C01789=1024.573,0.095,-96.896,167.247,47.803,158.792
C01790=1024.568,-0.154,-96.882,167.244,47.807,158.792
C01791=1024.561,-0.404,-96.867,167.241,47.810,158.792
C01792=1024.555,-0.653,-96.854,167.239,47.813,158.792
C01793=1024.549,-0.902,-96.839,167.236,47.817,158.792
C01794=1024.543,-1.152,-96.825,167.234,47.820,158.793
C01795=1024.538,-1.401,-96.810,167.231,47.823,158.793
C01796=1024.532,-1.652,-96.796,167.228,47.826,158.793
C01797=1024.526,-1.901,-96.782,167.226,47.830,158.794
C01798=1024.520,-2.150,-96.768,167.223,47.833,158.794
C01799=1024.514,-2.400,-96.753,167.221,47.836,158.794
C01800=1024.508,-2.649,-96.739,167.218,47.840,158.794
C01801=1024.502,-2.899,-96.726,167.214,47.843,158.794
C01802=1024.496,-3.148,-96.711,167.212,47.846,158.795
C01803=1024.490,-3.398,-96.697,167.209,47.850,158.795
C01804=1024.484,-3.648,-96.683,167.206,47.853,158.795
C01805=1024.478,-3.897,-96.668,167.204,47.856,158.795
C01806=1024.473,-4.147,-96.654,167.201,47.860,158.796
C01807=1024.466,-4.429,-96.639,167.198,47.863,158.796
C01808=1024.458,-4.711,-96.623,167.196,47.867,158.796
C01809=1024.452,-4.993,-96.608,167.193,47.871,158.797
C01810=1024.444,-5.274,-96.592,167.189,47.875,158.797
C01811=1024.439,-5.524,-96.578,167.187,47.878,158.797
C01812=1024.433,-5.774,-96.564,167.184,47.882,158.797
C01813=1024.426,-6.024,-96.550,167.181,47.885,158.798
C01814=1024.421,-6.272,-96.536,167.179,47.889,158.798
C01815=1024.414,-6.522,-96.522,167.176,47.892,158.798
C01816=1024.408,-6.772,-96.508,167.173,47.896,158.798
C01817=1024.402,-7.021,-96.495,167.169,47.899,158.799
C01818=1024.397,-7.271,-96.481,167.168,47.903,158.799
C01819=1024.389,-7.520,-96.467,167.164,47.906,158.799
C01820=1024.384,-7.770,-96.453,167.162,47.910,158.800
C01821=1024.378,-8.019,-96.439,167.159,47.912,158.800
C01822=1024.372,-8.269,-96.425,167.157,47.916,158.800
C01823=1024.366,-8.519,-96.412,167.153,47.919,158.800
C01824=1024.360,-8.768,-96.398,167.151,47.923,158.801
C01825=1024.353,-9.018,-96.384,167.148,47.926,158.801
C01826=1024.348,-9.268,-96.371,167.146,47.930,158.801
C01827=1024.341,-9.516,-96.357,167.142,47.933,158.801
C01828=1024.336,-9.766,-96.343,167.141,47.937,158.802
C01829=1024.329,-10.016,-96.329,167.137,47.940,158.802
C01830=1024.323,-10.265,-96.315,167.134,47.943,158.802
C01831=1024.317,-10.515,-96.302,167.132,47.947,158.802
C01832=1024.312,-10.764,-96.288,167.129,47.950,158.802
C01833=1024.305,-11.014,-96.274,167.126,47.954,158.803
C01834=1024.299,-11.264,-96.261,167.123,47.957,158.803
C01835=1024.293,-11.513,-96.247,167.121,47.960,158.803
C01836=1024.288,-11.763,-96.233,167.118,47.964,158.804
C01837=1024.281,-12.013,-96.220,167.115,47.967,158.804
C01838=1024.275,-12.262,-96.206,167.113,47.970,158.804
C01839=1024.269,-12.511,-96.193,167.110,47.974,158.804
C01840=1024.264,-12.761,-96.179,167.107,47.977,158.805
C01841=1024.258,-13.010,-96.166,167.105,47.980,158.805
C01842=1024.252,-13.261,-96.151,167.102,47.984,158.805
C01843=1024.245,-13.510,-96.138,167.099,47.987,158.805
C01844=1024.240,-13.759,-96.124,167.096,47.991,158.805
C01845=1024.234,-14.009,-96.111,167.094,47.994,158.806
C01846=1024.228,-14.258,-96.097,167.091,47.997,158.806
C01847=1024.221,-14.508,-96.083,167.088,48.000,158.806
C01848=1024.216,-14.758,-96.070,167.086,48.004,158.806
C01849=1024.210,-15.007,-96.056,167.083,48.007,158.807
C01850=1024.204,-15.257,-96.042,167.080,48.011,158.807
C01851=1024.198,-15.506,-96.029,167.078,48.014,158.807
C01852=1024.192,-15.755,-96.015,167.074,48.017,158.807
C01853=1024.186,-16.005,-96.002,167.072,48.021,158.808
C01854=1024.180,-16.255,-95.989,167.068,48.024,158.808
C01855=1024.174,-16.505,-95.976,167.067,48.028,158.808
C01856=1024.167,-16.754,-95.963,167.063,48.031,158.808
C01857=1024.162,-17.003,-95.949,167.060,48.035,158.809
C01858=1024.156,-17.253,-95.935,167.057,48.038,158.809
C01859=1024.149,-17.503,-95.923,167.054,48.042,158.809
C01860=1024.143,-17.753,-95.909,167.052,48.045,158.809
C01861=1024.137,-18.002,-95.895,167.049,48.049,158.810
C01862=1024.131,-18.251,-95.882,167.046,48.052,158.810
C01863=1024.125,-18.501,-95.870,167.043,48.056,158.810
C01864=1024.119,-18.751,-95.856,167.041,48.059,158.810
C01865=1024.113,-19.000,-95.843,167.038,48.062,158.811
C01866=1024.107,-19.249,-95.829,167.035,48.066,158.811
C01867=1024.101,-19.500,-95.816,167.032,48.070,158.811
C01868=1024.095,-19.749,-95.803,167.030,48.072,158.811
C01869=1024.088,-19.998,-95.790,167.027,48.076,158.812
C01870=1024.083,-20.248,-95.777,167.024,48.079,158.812
C01871=1024.076,-20.529,-95.762,167.021,48.083,158.812
C01872=1024.069,-20.809,-95.747,167.019,48.087,158.812
C01873=1024.062,-21.089,-95.732,167.015,48.091,158.813
C01874=1024.056,-21.369,-95.717,167.012,48.095,158.813
C01875=1024.050,-21.619,-95.704,167.009,48.098,158.813
C01876=1024.044,-21.868,-95.691,167.007,48.102,158.813
C01877=1024.037,-22.118,-95.678,167.004,48.105,158.814
C01878=1024.032,-22.368,-95.665,167.001,48.109,158.814
C01879=1024.026,-22.617,-95.651,166.998,48.112,158.814
C01880=1024.020,-22.866,-95.638,166.994,48.115,158.814
C01881=1024.014,-23.116,-95.626,166.993,48.119,158.815
C01882=1024.008,-23.366,-95.612,166.989,48.122,158.815
C01883=1024.002,-23.616,-95.600,166.987,48.126,158.815
C01884=1023.996,-23.865,-95.586,166.983,48.129,158.815
C01885=1023.990,-24.115,-95.573,166.981,48.132,158.815
C01886=1023.984,-24.364,-95.560,166.978,48.136,158.816
C01887=1023.978,-24.613,-95.547,166.975,48.139,158.816
C01888=1023.972,-24.863,-95.534,166.972,48.143,158.816
C01889=1023.967,-25.113,-95.520,166.970,48.146,158.816
C01890=1023.961,-25.363,-95.508,166.967,48.149,158.817
C01891=1023.954,-25.612,-95.494,166.964,48.153,158.817
C01892=1023.949,-25.862,-95.482,166.961,48.156,158.817
C01893=1023.942,-26.111,-95.469,166.959,48.159,158.817
C01894=1023.937,-26.361,-95.456,166.956,48.163,158.818
C01895=1023.931,-26.611,-95.442,166.953,48.166,158.818
C01896=1023.925,-26.861,-95.430,166.950,48.170,158.818
C01897=1023.919,-27.110,-95.416,166.948,48.173,158.818
C01898=1023.913,-27.360,-95.404,166.945,48.176,158.818
C01899=1023.907,-27.609,-95.391,166.942,48.180,158.819
C01900=1023.901,-27.859,-95.378,166.939,48.183,158.819
C01901=1023.895,-28.107,-95.365,166.936,48.187,158.819
C01902=1023.889,-28.357,-95.353,166.933,48.190,158.819
C01903=1023.883,-28.607,-95.340,166.931,48.194,158.820
C01904=1023.877,-28.856,-95.327,166.928,48.197,158.820
C01905=1023.871,-29.106,-95.314,166.925,48.201,158.820
C01906=1023.865,-29.356,-95.302,166.922,48.204,158.820
C01907=1023.859,-29.605,-95.288,166.919,48.208,158.821
C01908=1023.852,-29.855,-95.276,166.916,48.211,158.821
C01909=1023.847,-30.105,-95.264,166.914,48.215,158.821
C01910=1023.841,-30.355,-95.251,166.911,48.218,158.821
C01911=1023.834,-30.604,-95.238,166.908,48.222,158.822
C01912=1023.829,-30.854,-95.225,166.905,48.225,158.822
C01913=1023.823,-31.104,-95.213,166.902,48.229,158.822
C01914=1023.817,-31.352,-95.200,166.899,48.232,158.822
C01915=1023.811,-31.602,-95.187,166.897,48.236,158.822
C01916=1023.805,-31.852,-95.175,166.894,48.239,158.823
C01917=1023.799,-32.102,-95.162,166.891,48.243,158.823
C01918=1023.792,-32.351,-95.150,166.888,48.246,158.823
C01919=1023.786,-32.601,-95.137,166.885,48.250,158.823
C01920=1023.781,-32.851,-95.125,166.882,48.253,158.824
C01921=1023.775,-33.100,-95.112,166.880,48.257,158.824
C01922=1023.769,-33.350,-95.100,166.877,48.260,158.824
C01923=1023.763,-33.599,-95.087,166.874,48.263,158.824
C01924=1023.757,-33.849,-95.074,166.871,48.267,158.824
C01925=1023.751,-34.099,-95.061,166.868,48.270,158.825
C01926=1023.745,-34.349,-95.049,166.865,48.274,158.825
C01927=1023.739,-34.598,-95.037,166.863,48.277,158.825
C01928=1023.733,-34.847,-95.024,166.860,48.281,158.825
C01929=1023.727,-35.097,-95.012,166.857,48.284,158.826
C01930=1023.721,-35.347,-94.999,166.853,48.288,158.826
C01931=1023.715,-35.597,-94.986,166.851,48.291,158.826
C01932=1023.710,-35.846,-94.974,166.847,48.295,158.826
C01933=1023.704,-36.096,-94.962,166.846,48.298,158.827
C01934=1023.698,-36.346,-94.949,166.842,48.302,158.827
C01935=1023.691,-36.625,-94.935,166.840,48.305,158.827
C01936=1023.685,-36.904,-94.921,166.836,48.310,158.827
C01937=1023.678,-37.184,-94.907,166.833,48.313,158.827
C01938=1023.671,-37.463,-94.893,166.830,48.317,158.828
C01939=1023.666,-37.712,-94.881,166.827,48.320,158.828
C01940=1023.660,-37.962,-94.869,166.824,48.324,158.828
C01941=1023.654,-38.212,-94.856,166.821,48.327,158.828
C01942=1023.648,-38.462,-94.844,166.818,48.331,158.828
C01943=1023.643,-38.711,-94.831,166.816,48.334,158.829
C01944=1023.636,-38.961,-94.819,166.812,48.337,158.829
C01945=1023.630,-39.210,-94.807,166.810,48.341,158.829
C01946=1023.624,-39.460,-94.794,166.806,48.344,158.829
C01947=1023.618,-39.709,-94.783,166.804,48.348,158.830
C01948=1023.612,-39.959,-94.770,166.800,48.351,158.830
C01949=1023.607,-40.209,-94.758,166.798,48.355,158.830
C01950=1023.600,-40.459,-94.746,166.794,48.358,158.830
C01951=1023.595,-40.708,-94.733,166.793,48.362,158.831
C01952=1023.589,-40.958,-94.721,166.789,48.365,158.831
C01953=1023.582,-41.207,-94.709,166.787,48.369,158.831
C01954=1023.577,-41.457,-94.697,166.783,48.372,158.831
C01955=1023.570,-41.707,-94.685,166.781,48.376,158.831
C01956=1023.565,-41.956,-94.673,166.777,48.379,158.832
C01957=1023.559,-42.206,-94.661,166.775,48.383,158.832
C01958=1023.553,-42.455,-94.649,166.771,48.387,158.832
C01959=1023.547,-42.705,-94.636,166.769,48.390,158.832
C01960=1023.541,-42.955,-94.625,166.765,48.394,158.832
C01961=1023.535,-43.204,-94.613,166.764,48.397,158.833
C01962=1023.529,-43.454,-94.600,166.761,48.401,158.833
C01963=1023.523,-43.703,-94.589,166.758,48.404,158.833
C01964=1023.517,-43.953,-94.576,166.755,48.408,158.833
C01965=1023.511,-44.203,-94.565,166.752,48.412,158.834
C01966=1023.505,-44.452,-94.553,166.749,48.415,158.834
C01967=1023.500,-44.702,-94.540,166.746,48.419,158.834
C01968=1023.493,-44.952,-94.528,166.743,48.422,158.834
C01969=1023.488,-45.202,-94.517,166.739,48.425,158.834
C01970=1023.481,-45.451,-94.505,166.737,48.429,158.835
C01971=1023.476,-45.700,-94.493,166.734,48.432,158.835
C01972=1023.470,-45.950,-94.480,166.732,48.436,158.835
C01973=1023.464,-46.201,-94.469,166.728,48.439,158.835
C01974=1023.458,-46.450,-94.457,166.726,48.443,158.836
C01975=1023.452,-46.699,-94.445,166.722,48.446,158.836
C01976=1023.447,-46.949,-94.433,166.719,48.449,158.836
C01977=1023.440,-47.199,-94.421,166.716,48.453,158.836
C01978=1023.435,-47.448,-94.409,166.713,48.457,158.836
C01979=1023.429,-47.698,-94.396,166.710,48.461,158.837
C01980=1023.423,-47.947,-94.386,166.708,48.463,158.837
C01981=1023.417,-48.197,-94.373,166.705,48.467,158.837
C01982=1023.411,-48.447,-94.362,166.702,48.471,158.837
C01983=1023.406,-48.696,-94.350,166.699,48.474,158.837
C01984=1023.399,-48.946,-94.338,166.696,48.478,158.838
C01985=1023.394,-49.196,-94.326,166.693,48.481,158.838
C01986=1023.388,-49.446,-94.314,166.690,48.484,158.838
C01987=1023.382,-49.695,-94.302,166.687,48.488,158.838
C01988=1023.376,-49.945,-94.290,166.684,48.491,158.838
C01989=1023.370,-50.194,-94.279,166.682,48.494,158.839
C01990=1023.365,-50.444,-94.267,166.679,48.498,158.839
C01991=1023.359,-50.693,-94.255,166.676,48.501,158.839
C01992=1023.353,-50.944,-94.243,166.673,48.505,158.839
C01993=1023.347,-51.193,-94.232,166.670,48.509,158.839
C01994=1023.341,-51.443,-94.220,166.667,48.512,158.840
C01995=1023.335,-51.692,-94.209,166.664,48.516,158.840
C01996=1023.329,-51.942,-94.197,166.661,48.520,158.840
C01997=1023.323,-52.192,-94.186,166.658,48.524,158.840
C01998=1023.317,-52.441,-94.174,166.655,48.527,158.840
C01999=1023.310,-52.722,-94.162,166.652,48.532,158.841
C02000=1023.303,-53.001,-94.149,166.649,48.536,158.841
C02001=1023.297,-53.280,-94.136,166.645,48.540,158.841
C02002=1023.290,-53.561,-94.124,166.642,48.544,158.842
C02003=1023.284,-53.810,-94.112,166.639,48.547,158.842
C02004=1023.278,-54.060,-94.101,166.636,48.551,158.842
C02005=1023.272,-54.310,-94.089,166.633,48.554,158.842
C02006=1023.266,-54.559,-94.077,166.630,48.558,158.842
C02007=1023.261,-54.809,-94.066,166.627,48.562,158.843
C02008=1023.254,-55.059,-94.055,166.624,48.565,158.843
C02009=1023.248,-55.308,-94.044,166.621,48.569,158.843
C02010=1023.242,-55.558,-94.032,166.618,48.572,158.843
C02011=1023.236,-55.807,-94.021,166.615,48.576,158.844
C02012=1023.230,-56.058,-94.010,166.613,48.580,158.844
C02013=1023.224,-56.307,-93.998,166.609,48.583,158.844
C02014=1023.219,-56.556,-93.987,166.607,48.587,158.844
C02015=1023.212,-56.806,-93.976,166.603,48.591,158.844
C02016=1023.207,-57.056,-93.965,166.601,48.595,158.845
C02017=1023.200,-57.305,-93.953,166.597,48.598,158.845
C02018=1023.195,-57.555,-93.942,166.595,48.602,158.845
C02019=1023.189,-57.805,-93.931,166.591,48.605,158.845
C02020=1023.183,-58.055,-93.919,166.589,48.609,158.846
C02021=1023.177,-58.304,-93.908,166.585,48.612,158.846
C02022=1023.171,-58.553,-93.897,166.583,48.616,158.846
C02023=1023.165,-58.803,-93.886,166.580,48.620,158.846
C02024=1023.159,-59.053,-93.875,166.577,48.623,158.846
C02025=1023.153,-59.303,-93.863,166.574,48.627,158.847
C02026=1023.148,-59.553,-93.852,166.571,48.630,158.847
C02027=1023.142,-59.802,-93.841,166.568,48.634,158.847
C02028=1023.136,-60.051,-93.830,166.565,48.638,158.847
C02029=1023.130,-60.301,-93.818,166.562,48.642,158.847
C02030=1023.124,-60.551,-93.808,166.559,48.645,158.848
C02031=1023.118,-60.800,-93.797,166.556,48.649,158.848
C02032=1023.112,-61.051,-93.785,166.553,48.652,158.848
C02033=1023.107,-61.300,-93.774,166.550,48.656,158.848
C02034=1023.101,-61.550,-93.763,166.547,48.659,158.848
C02035=1023.095,-61.800,-93.752,166.544,48.663,158.849
C02036=1023.089,-62.050,-93.741,166.541,48.666,158.849
///RCONF 1,0,0,1,0,0,0,0,0,0,0,0,0,0,0,0,0,0,0,0,0,0,0,0
C02037=1023.083,-62.298,-93.729,166.538,48.670,158.849
C02038=1023.077,-62.548,-93.719,166.535,48.674,158.849
C02039=1023.072,-62.798,-93.707,166.532,48.677,158.849
C02040=1023.066,-63.048,-93.696,166.529,48.681,158.850
C02041=1023.060,-63.297,-93.685,166.526,48.684,158.850
C02042=1023.054,-63.547,-93.674,166.523,48.688,158.850
C02043=1023.048,-63.797,-93.663,166.520,48.691,158.850
C02044=1023.042,-64.047,-93.652,166.517,48.695,158.850
C02045=1023.036,-64.296,-93.641,166.514,48.698,158.851
C02046=1023.031,-64.546,-93.630,166.511,48.702,158.851
C02047=1023.025,-64.796,-93.618,166.508,48.705,158.851
C02048=1023.019,-65.046,-93.607,166.505,48.709,158.851
C02049=1023.014,-65.295,-93.597,166.502,48.713,158.851
C02050=1023.008,-65.545,-93.586,166.499,48.716,158.851
C02051=1023.002,-65.794,-93.575,166.496,48.720,158.852
C02052=1022.996,-66.044,-93.564,166.493,48.723,158.852
C02053=1022.990,-66.294,-93.553,166.490,48.727,158.852
C02054=1022.985,-66.544,-93.543,166.487,48.730,158.852
C02055=1022.980,-66.794,-93.531,166.484,48.734,158.852
C02056=1022.974,-67.043,-93.520,166.481,48.738,158.853
C02057=1022.968,-67.293,-93.509,166.478,48.741,158.853
C02058=1022.962,-67.542,-93.498,166.475,48.745,158.853
C02059=1022.956,-67.792,-93.487,166.472,48.748,158.853
C02060=1022.950,-68.042,-93.476,166.470,48.751,158.853
C02061=1022.945,-68.291,-93.465,166.467,48.755,158.854
C02062=1022.939,-68.541,-93.455,166.464,48.758,158.854
C02063=1022.933,-68.822,-93.443,166.460,48.762,158.854
C02064=1022.926,-69.104,-93.430,166.457,48.766,158.854
C02065=1022.920,-69.384,-93.418,166.453,48.771,158.854
C02066=1022.914,-69.665,-93.406,166.450,48.774,158.855
C02067=1022.908,-69.914,-93.395,166.447,48.778,158.855
C02068=1022.902,-70.164,-93.384,166.444,48.781,158.855
C02069=1022.896,-70.413,-93.374,166.441,48.785,158.855
C02070=1022.891,-70.663,-93.362,166.438,48.788,158.855
C02071=1022.886,-70.913,-93.352,166.435,48.791,158.855
C02072=1022.880,-71.163,-93.341,166.432,48.795,158.856
C02073=1022.874,-71.413,-93.330,166.429,48.799,158.856
C02074=1022.868,-71.662,-93.319,166.426,48.802,158.856
C02075=1022.863,-71.913,-93.309,166.423,48.806,158.856
C02076=1022.857,-72.162,-93.298,166.420,48.809,158.856
C02077=1022.851,-72.412,-93.287,166.417,48.812,158.856
C02078=1022.845,-72.661,-93.276,166.414,48.816,158.857
C02079=1022.840,-72.911,-93.266,166.411,48.820,158.857
C02080=1022.834,-73.161,-93.255,166.408,48.823,158.857
C02081=1022.829,-73.410,-93.244,166.405,48.827,158.857
C02082=1022.824,-73.660,-93.233,166.402,48.830,158.857
C02083=1022.818,-73.910,-93.223,166.398,48.833,158.857
C02084=1022.812,-74.160,-93.212,166.396,48.837,158.858
C02085=1022.807,-74.410,-93.202,166.394,48.840,158.858
C02086=1022.801,-74.659,-93.191,166.389,48.844,158.858
C02087=1022.795,-74.908,-93.180,166.387,48.848,158.858
C02088=1022.789,-75.158,-93.170,166.383,48.851,158.858
C02089=1022.784,-75.408,-93.159,166.381,48.855,158.859
C02090=1022.778,-75.658,-93.149,166.377,48.858,158.859
C02091=1022.772,-75.907,-93.139,166.375,48.862,158.859
C02092=1022.766,-76.157,-93.129,166.371,48.865,158.859
C02093=1022.760,-76.407,-93.118,166.369,48.869,158.859
C02094=1022.755,-76.657,-93.108,166.366,48.873,158.860
C02095=1022.749,-76.906,-93.097,166.363,48.877,158.860
C02096=1022.743,-77.156,-93.087,166.360,48.880,158.860
C02097=1022.737,-77.406,-93.076,166.357,48.884,158.860
C02098=1022.732,-77.656,-93.066,166.354,48.887,158.860
C02099=1022.726,-77.905,-93.055,166.351,48.891,158.861
C02100=1022.721,-78.155,-93.045,166.348,48.894,158.861
C02101=1022.715,-78.405,-93.036,166.345,48.898,158.861
C02102=1022.709,-78.654,-93.025,166.342,48.902,158.861
C02103=1022.704,-78.904,-93.015,166.339,48.906,158.861
C02104=1022.698,-79.154,-93.004,166.336,48.909,158.861
C02105=1022.692,-79.403,-92.994,166.333,48.913,158.862
C02106=1022.686,-79.653,-92.984,166.330,48.916,158.862
C02107=1022.681,-79.903,-92.973,166.327,48.920,158.862
C02108=1022.676,-80.153,-92.963,166.324,48.923,158.862
C02109=1022.669,-80.402,-92.953,166.320,48.928,158.862
C02110=1022.664,-80.652,-92.943,166.317,48.931,158.863
C02111=1022.657,-80.902,-92.933,166.314,48.935,158.863
C02112=1022.652,-81.152,-92.923,166.311,48.939,158.863
C02113=1022.646,-81.401,-92.913,166.308,48.942,158.863
C02114=1022.641,-81.651,-92.903,166.305,48.946,158.863
C02115=1022.635,-81.901,-92.893,166.302,48.949,158.864
C02116=1022.629,-82.151,-92.883,166.299,48.953,158.864
C02117=1022.623,-82.401,-92.874,166.297,48.957,158.864
C02118=1022.617,-82.650,-92.863,166.292,48.961,158.864
C02119=1022.611,-82.900,-92.853,166.290,48.965,158.864
C02120=1022.606,-83.149,-92.844,166.286,48.968,158.864
C02121=1022.600,-83.399,-92.834,166.284,48.972,158.865
C02122=1022.595,-83.649,-92.824,166.281,48.976,158.865
C02123=1022.588,-83.898,-92.813,166.278,48.979,158.865
C02124=1022.583,-84.148,-92.803,166.275,48.983,158.865
C02125=1022.576,-84.398,-92.794,166.272,48.987,158.866
C02126=1022.572,-84.648,-92.784,166.269,48.991,158.866
C02127=1022.565,-84.931,-92.773,166.265,48.995,158.866
C02128=1022.558,-85.214,-92.762,166.261,48.999,158.866
C02129=1022.551,-85.497,-92.751,166.258,49.003,158.866
C02130=1022.546,-85.780,-92.739,166.255,49.007,158.867
C02131=1022.539,-86.030,-92.729,166.252,49.011,158.867
C02132=1022.534,-86.280,-92.719,166.249,49.015,158.867
C02133=1022.528,-86.529,-92.710,166.246,49.019,158.867
C02134=1022.523,-86.779,-92.700,166.243,49.022,158.867
C02135=1022.517,-87.029,-92.690,166.239,49.026,158.868
C02136=1022.511,-87.279,-92.680,166.236,49.030,158.868
C02137=1022.506,-87.528,-92.671,166.233,49.033,158.868
C02138=1022.500,-87.778,-92.661,166.230,49.037,158.868
C02139=1022.494,-88.028,-92.651,166.227,49.041,158.868
C02140=1022.488,-88.278,-92.641,166.224,49.045,158.869
C02141=1022.483,-88.527,-92.632,166.221,49.048,158.869
C02142=1022.477,-88.777,-92.622,166.218,49.052,158.869
C02143=1022.472,-89.027,-92.612,166.215,49.055,158.869
C02144=1022.466,-89.276,-92.603,166.212,49.059,158.869
C02145=1022.461,-89.526,-92.593,166.209,49.062,158.869
C02146=1022.454,-89.776,-92.583,166.205,49.067,158.870
C02147=1022.449,-90.026,-92.573,166.202,49.070,158.870
C02148=1022.443,-90.275,-92.564,166.199,49.074,158.870
C02149=1022.438,-90.525,-92.553,166.196,49.077,158.870
C02150=1022.432,-90.775,-92.544,166.193,49.081,158.870
C02151=1022.427,-91.024,-92.534,166.190,49.085,158.870
C02152=1022.421,-91.274,-92.525,166.188,49.089,158.871
C02153=1022.415,-91.524,-92.514,166.184,49.092,158.871
C02154=1022.410,-91.773,-92.505,166.182,49.096,158.871
C02155=1022.404,-92.024,-92.496,166.178,49.099,158.871
C02156=1022.399,-92.273,-92.487,166.176,49.103,158.871
C02157=1022.393,-92.523,-92.477,166.173,49.106,158.871
C02158=1022.387,-92.773,-92.467,166.170,49.110,158.872
C02159=1022.382,-93.022,-92.458,166.166,49.114,158.872
C02160=1022.376,-93.272,-92.447,166.163,49.118,158.872
C02161=1022.371,-93.521,-92.438,166.160,49.121,158.872
C02162=1022.365,-93.772,-92.428,166.157,49.125,158.872
C02163=1022.360,-94.022,-92.419,166.154,49.129,158.872
C02164=1022.354,-94.271,-92.410,166.151,49.133,158.873
C02165=1022.349,-94.521,-92.400,166.148,49.136,158.873
C02166=1022.343,-94.770,-92.391,166.145,49.140,158.873
C02167=1022.338,-95.020,-92.381,166.142,49.143,158.873
C02168=1022.332,-95.270,-92.372,166.139,49.146,158.873
C02169=1022.327,-95.520,-92.362,166.136,49.150,158.874
C02170=1022.321,-95.770,-92.352,166.133,49.154,158.874
C02171=1022.316,-96.019,-92.343,166.130,49.158,158.874
C02172=1022.310,-96.270,-92.334,166.127,49.161,158.874
C02173=1022.304,-96.519,-92.324,166.124,49.165,158.874
C02174=1022.299,-96.769,-92.314,166.121,49.168,158.874
C02175=1022.293,-97.018,-92.305,166.117,49.172,158.874
C02176=1022.288,-97.269,-92.296,166.114,49.176,158.875
C02177=1022.283,-97.518,-92.286,166.111,49.179,158.875
C02178=1022.277,-97.768,-92.276,166.108,49.183,158.875
C02179=1022.272,-98.018,-92.268,166.105,49.186,158.875
C02180=1022.266,-98.268,-92.258,166.102,49.190,158.875
C02181=1022.260,-98.517,-92.249,166.099,49.194,158.876
C02182=1022.254,-98.767,-92.240,166.096,49.198,158.876
C02183=1022.249,-99.016,-92.231,166.093,49.202,158.876
C02184=1022.244,-99.267,-92.222,166.089,49.205,158.876
C02185=1022.238,-99.516,-92.212,166.086,49.209,158.876
C02186=1022.232,-99.766,-92.203,166.084,49.213,158.877
C02187=1022.227,-100.016,-92.194,166.081,49.217,158.877
C02188=1022.221,-100.266,-92.185,166.078,49.221,158.877
C02189=1022.215,-100.515,-92.176,166.075,49.224,158.877
C02190=1022.209,-100.765,-92.167,166.072,49.228,158.877
C02191=1022.204,-101.050,-92.157,166.068,49.232,158.877
C02192=1022.197,-101.336,-92.147,166.064,49.237,158.878
C02193=1022.191,-101.620,-92.136,166.061,49.241,158.878
C02194=1022.184,-101.906,-92.126,166.058,49.245,158.878
C02195=1022.179,-102.155,-92.116,166.055,49.249,158.878
C02196=1022.174,-102.405,-92.108,166.052,49.252,158.878
C02197=1022.168,-102.655,-92.098,166.048,49.256,158.879
C02198=1022.163,-102.904,-92.090,166.045,49.260,158.879
C02199=1022.156,-103.154,-92.080,166.042,49.264,158.879
C02200=1022.151,-103.404,-92.071,166.039,49.268,158.879
C02201=1022.146,-103.654,-92.063,166.036,49.271,158.879
C02202=1022.140,-103.904,-92.053,166.033,49.275,158.879
C02203=1022.135,-104.153,-92.044,166.030,49.278,158.880
C02204=1022.129,-104.403,-92.035,166.027,49.282,158.880
C02205=1022.124,-104.653,-92.026,166.024,49.286,158.880
C02206=1022.118,-104.903,-92.018,166.020,49.290,158.880
C02207=1022.112,-105.152,-92.008,166.017,49.294,158.880
C02208=1022.107,-105.402,-92.000,166.014,49.297,158.880
C02209=1022.102,-105.652,-91.991,166.012,49.301,158.881
C02210=1022.096,-105.902,-91.982,166.008,49.305,158.881
C02211=1022.091,-106.152,-91.973,166.006,49.309,158.881
C02212=1022.086,-106.401,-91.964,166.003,49.312,158.881
C02213=1022.080,-106.651,-91.955,166.000,49.316,158.881
C02214=1022.074,-106.901,-91.946,165.996,49.320,158.881
C02215=1022.069,-107.151,-91.938,165.993,49.324,158.882
C02216=1022.063,-107.401,-91.929,165.990,49.328,158.882
C02217=1022.058,-107.650,-91.920,165.987,49.331,158.882
C02218=1022.052,-107.900,-91.911,165.984,49.335,158.882
C02219=1022.047,-108.150,-91.902,165.981,49.338,158.882
C02220=1022.041,-108.400,-91.894,165.978,49.342,158.883
C02221=1022.036,-108.650,-91.885,165.975,49.346,158.883
C02222=1022.030,-108.899,-91.876,165.971,49.350,158.883
C02223=1022.025,-109.149,-91.867,165.968,49.354,158.883
C02224=1022.019,-109.399,-91.859,165.965,49.357,158.883
C02225=1022.013,-109.648,-91.851,165.963,49.361,158.883
C02226=1022.008,-109.898,-91.842,165.960,49.365,158.884
C02227=1022.002,-110.149,-91.833,165.957,49.369,158.884
C02228=1021.997,-110.398,-91.824,165.953,49.373,158.884
C02229=1021.991,-110.647,-91.816,165.950,49.377,158.884
C02230=1021.986,-110.897,-91.807,165.947,49.380,158.884
C02231=1021.980,-111.147,-91.798,165.944,49.384,158.885
C02232=1021.975,-111.397,-91.790,165.941,49.388,158.885
C02233=1021.970,-111.647,-91.781,165.938,49.392,158.885
C02234=1021.964,-111.897,-91.773,165.935,49.396,158.885
C02235=1021.959,-112.146,-91.765,165.932,49.399,158.885
C02236=1021.953,-112.397,-91.756,165.928,49.403,158.885
C02237=1021.947,-112.646,-91.748,165.925,49.407,158.885
C02238=1021.942,-112.896,-91.739,165.923,49.411,158.886
C02239=1021.937,-113.146,-91.731,165.919,49.414,158.886
C02240=1021.931,-113.395,-91.722,165.917,49.418,158.886
C02241=1021.926,-113.646,-91.713,165.914,49.422,158.886
C02242=1021.920,-113.895,-91.705,165.911,49.425,158.886
C02243=1021.915,-114.145,-91.697,165.907,49.430,158.887
C02244=1021.910,-114.395,-91.688,165.904,49.433,158.887
C02245=1021.905,-114.645,-91.680,165.901,49.437,158.887
C02246=1021.899,-114.894,-91.672,165.898,49.441,158.887
C02247=1021.893,-115.144,-91.663,165.895,49.444,158.887
C02248=1021.887,-115.394,-91.654,165.892,49.448,158.888
C02249=1021.882,-115.644,-91.646,165.890,49.452,158.888
C02250=1021.877,-115.894,-91.637,165.885,49.456,158.888
C02251=1021.871,-116.143,-91.629,165.883,49.460,158.888
C02252=1021.866,-116.393,-91.621,165.879,49.463,158.888
C02253=1021.860,-116.642,-91.612,165.877,49.467,158.888
C02254=1021.855,-116.893,-91.605,165.874,49.471,158.889
C02255=1021.849,-117.178,-91.595,165.870,49.476,158.889
C02256=1021.843,-117.462,-91.586,165.866,49.480,158.889
C02257=1021.837,-117.747,-91.576,165.863,49.484,158.889
C02258=1021.830,-118.032,-91.567,165.860,49.488,158.889
C02259=1021.824,-118.282,-91.559,165.857,49.493,158.890
C02260=1021.819,-118.531,-91.550,165.854,49.497,158.890
C02261=1021.814,-118.782,-91.542,165.850,49.500,158.890
C02262=1021.809,-119.031,-91.534,165.847,49.504,158.890
C02263=1021.803,-119.281,-91.526,165.844,49.508,158.890
C02264=1021.798,-119.530,-91.518,165.841,49.512,158.890
C02265=1021.793,-119.781,-91.510,165.838,49.516,158.891
C02266=1021.787,-120.030,-91.502,165.835,49.519,158.891
C02267=1021.781,-120.280,-91.493,165.833,49.523,158.891
C02268=1021.776,-120.530,-91.485,165.829,49.527,158.891
C02269=1021.771,-120.780,-91.477,165.826,49.531,158.891
C02270=1021.765,-121.029,-91.469,165.823,49.535,158.891
C02271=1021.760,-121.279,-91.461,165.820,49.538,158.891
C02272=1021.755,-121.529,-91.453,165.817,49.542,158.892
C02273=1021.749,-121.779,-91.445,165.814,49.546,158.892
C02274=1021.744,-122.029,-91.437,165.811,49.549,158.892
C02275=1021.739,-122.279,-91.429,165.807,49.554,158.892
C02276=1021.733,-122.528,-91.421,165.804,49.558,158.892
C02277=1021.727,-122.778,-91.412,165.801,49.561,158.893
C02278=1021.722,-123.028,-91.405,165.799,49.565,158.893
C02279=1021.716,-123.278,-91.397,165.795,49.569,158.893
C02280=1021.711,-123.527,-91.388,165.793,49.573,158.893
C02281=1021.706,-123.778,-91.381,165.790,49.577,158.893
C02282=1021.700,-124.027,-91.373,165.787,49.580,158.893
C02283=1021.695,-124.278,-91.365,165.783,49.584,158.894
C02284=1021.690,-124.527,-91.356,165.780,49.588,158.894
C02285=1021.684,-124.777,-91.349,165.777,49.592,158.894
C02286=1021.679,-125.027,-91.341,165.774,49.596,158.894
C02287=1021.673,-125.276,-91.333,165.772,49.600,158.894
C02288=1021.668,-125.527,-91.325,165.768,49.603,158.895
C02289=1021.662,-125.776,-91.317,165.765,49.607,158.895
C02290=1021.658,-126.026,-91.310,165.762,49.612,158.895
C02291=1021.652,-126.276,-91.303,165.759,49.615,158.895
C02292=1021.647,-126.526,-91.294,165.756,49.619,158.895
C02293=1021.642,-126.776,-91.286,165.753,49.623,158.895
C02294=1021.636,-127.025,-91.278,165.750,49.626,158.896
C02295=1021.631,-127.276,-91.271,165.747,49.630,158.896
C02296=1021.625,-127.525,-91.263,165.743,49.635,158.896
C02297=1021.621,-127.775,-91.255,165.740,49.638,158.896
C02298=1021.615,-128.024,-91.248,165.738,49.642,158.896
C02299=1021.609,-128.274,-91.239,165.734,49.645,158.896
C02300=1021.605,-128.523,-91.230,165.732,49.648,158.897
C02301=1021.601,-128.773,-91.221,165.729,49.650,158.896
C02302=1021.598,-129.022,-91.211,165.726,49.653,158.896
C02303=1021.595,-129.272,-91.200,165.723,49.654,158.896
C02304=1021.592,-129.522,-91.189,165.721,49.655,158.896
C02305=1021.591,-129.772,-91.177,165.719,49.655,158.895
C02306=1021.589,-130.021,-91.165,165.716,49.655,158.895
C02307=1021.588,-130.271,-91.153,165.714,49.654,158.895
C02308=1021.587,-130.521,-91.138,165.711,49.653,158.894
C02309=1021.587,-130.771,-91.124,165.709,49.652,158.893
C02310=1021.588,-131.020,-91.110,165.707,49.649,158.893
C02311=1021.588,-131.270,-91.095,165.705,49.646,158.892
C02312=1021.590,-131.520,-91.078,165.703,49.644,158.891
C02313=1021.592,-131.770,-91.062,165.701,49.640,158.890
C02314=1021.594,-132.019,-91.046,165.700,49.635,158.889
C02315=1021.597,-132.269,-91.028,165.698,49.630,158.888
C02316=1021.600,-132.520,-91.009,165.696,49.625,158.887
C02317=1021.604,-132.769,-90.990,165.695,49.620,158.886
C02318=1021.608,-133.018,-90.971,165.693,49.614,158.884
C02319=1021.324,-133.044,-91.324,165.647,49.915,158.928
C02320=1021.321,-132.937,-91.332,165.648,49.918,158.929
C02321=1021.316,-132.580,-91.360,165.650,49.927,158.931
C02322=1021.313,-132.330,-91.378,165.651,49.932,158.932
C02323=1021.310,-132.080,-91.396,165.652,49.937,158.933
C02324=1021.308,-131.830,-91.413,165.655,49.941,158.934
C02325=1021.305,-131.580,-91.429,165.656,49.945,158.935
C02326=1021.304,-131.331,-91.445,165.659,49.948,158.936
C02327=1021.303,-131.081,-91.461,165.661,49.951,158.936
C02328=1021.302,-130.831,-91.475,165.663,49.953,158.937
C02329=1021.303,-130.581,-91.490,165.665,49.955,158.938
C02330=1021.304,-130.332,-91.503,165.667,49.956,158.938
C02331=1021.305,-130.082,-91.516,165.669,49.957,158.939
C02332=1021.305,-129.832,-91.528,165.672,49.957,158.939
C02333=1021.309,-129.420,-91.548,165.676,49.956,158.940
C02334=1021.313,-129.008,-91.565,165.680,49.954,158.940
C02335=1021.320,-128.596,-91.582,165.685,49.950,158.940
C02336=1021.327,-128.185,-91.596,165.690,49.946,158.940
C02337=1021.332,-127.935,-91.604,165.693,49.942,158.940
C02338=1021.338,-127.685,-91.612,165.696,49.938,158.940
C02339=1021.343,-127.435,-91.620,165.699,49.934,158.940
C02340=1021.348,-127.186,-91.627,165.701,49.930,158.939
C02341=1021.353,-126.936,-91.635,165.706,49.926,158.939
C02342=1021.359,-126.687,-91.643,165.708,49.922,158.939
C02343=1021.364,-126.436,-91.651,165.711,49.918,158.939
C02344=1021.370,-126.187,-91.658,165.714,49.914,158.939
C02345=1021.375,-125.936,-91.666,165.717,49.911,158.939
C02346=1021.381,-125.688,-91.674,165.721,49.906,158.939
C02347=1021.386,-125.437,-91.681,165.723,49.902,158.938
C02348=1021.391,-125.187,-91.689,165.726,49.898,158.938
C02349=1021.397,-124.938,-91.697,165.729,49.895,158.938
C02350=1021.402,-124.688,-91.704,165.732,49.891,158.938
C02351=1021.408,-124.438,-91.713,165.736,49.886,158.938
C02352=1021.413,-124.188,-91.721,165.739,49.883,158.938
C02353=1021.419,-123.938,-91.728,165.742,49.879,158.937
C02354=1021.424,-123.689,-91.737,165.744,49.875,158.937
C02355=1021.429,-123.438,-91.745,165.748,49.872,158.937
C02356=1021.434,-123.190,-91.752,165.750,49.868,158.937
C02357=1021.439,-122.939,-91.760,165.754,49.863,158.937
C02358=1021.444,-122.689,-91.768,165.757,49.860,158.936
C02359=1021.450,-122.440,-91.776,165.760,49.856,158.936
C02360=1021.455,-122.190,-91.784,165.763,49.852,158.936
C02361=1021.461,-121.940,-91.793,165.766,49.848,158.936
C02362=1021.467,-121.691,-91.801,165.769,49.844,158.936
C02363=1021.472,-121.440,-91.808,165.772,49.840,158.936
C02364=1021.477,-121.191,-91.817,165.775,49.837,158.935
C02365=1021.483,-120.941,-91.825,165.778,49.832,158.935
C02366=1021.488,-120.691,-91.832,165.781,49.828,158.935
C02367=1021.493,-120.441,-91.841,165.784,49.825,158.935
C02368=1021.499,-120.192,-91.849,165.787,49.821,158.935
C02369=1021.504,-119.941,-91.857,165.791,49.817,158.934
C02370=1021.509,-119.692,-91.865,165.794,49.813,158.934
C02371=1021.515,-119.442,-91.874,165.796,49.809,158.934
C02372=1021.521,-119.193,-91.881,165.799,49.805,158.934
C02373=1021.526,-118.942,-91.889,165.802,49.801,158.934
C02374=1021.531,-118.692,-91.898,165.806,49.797,158.934
C02375=1021.536,-118.443,-91.906,165.809,49.793,158.933
C02376=1021.542,-118.193,-91.914,165.812,49.789,158.933
C02377=1021.549,-117.874,-91.924,165.815,49.785,158.933
C02378=1021.556,-117.555,-91.935,165.820,49.779,158.933
C02379=1021.563,-117.238,-91.945,165.823,49.774,158.933
C02380=1021.570,-116.919,-91.956,165.827,49.770,158.932
C02381=1021.575,-116.669,-91.965,165.831,49.766,158.932
C02382=1021.580,-116.419,-91.972,165.834,49.762,158.932
C02383=1021.586,-116.170,-91.980,165.837,49.758,158.932
C02384=1021.591,-115.920,-91.989,165.839,49.754,158.932
C02385=1021.596,-115.670,-91.997,165.842,49.750,158.931
C02386=1021.602,-115.420,-92.006,165.845,49.747,158.931
C02387=1021.608,-115.171,-92.014,165.849,49.742,158.931
C02388=1021.614,-114.921,-92.023,165.852,49.738,158.931
C02389=1021.619,-114.671,-92.031,165.855,49.734,158.931
C02390=1021.624,-114.421,-92.040,165.858,49.731,158.931
C02391=1021.629,-114.171,-92.047,165.860,49.727,158.930
C02392=1021.634,-113.921,-92.056,165.865,49.723,158.930
C02393=1021.640,-113.671,-92.064,165.867,49.719,158.930
C02394=1021.645,-113.422,-92.073,165.870,49.715,158.930
C02395=1021.651,-113.172,-92.081,165.873,49.712,158.930
C02396=1021.657,-112.922,-92.089,165.876,49.708,158.929
C02397=1021.662,-112.672,-92.098,165.879,49.704,158.929
C02398=1021.667,-112.422,-92.106,165.883,49.700,158.929
C02399=1021.672,-112.173,-92.115,165.886,49.696,158.929
C02400=1021.678,-111.924,-92.124,165.888,49.692,158.929
C02401=1021.684,-111.673,-92.133,165.892,49.689,158.929
C02402=1021.689,-111.423,-92.141,165.894,49.685,158.928
C02403=1021.694,-111.174,-92.150,165.897,49.681,158.928
C02404=1021.700,-110.924,-92.158,165.901,49.677,158.928
C02405=1021.705,-110.674,-92.167,165.904,49.673,158.928
C02406=1021.712,-110.424,-92.175,165.907,49.669,158.928
C02407=1021.717,-110.175,-92.184,165.910,49.665,158.928
C02408=1021.722,-109.925,-92.192,165.913,49.661,158.927
C02409=1021.727,-109.675,-92.201,165.916,49.657,158.927
C02410=1021.733,-109.425,-92.209,165.919,49.654,158.927
C02411=1021.739,-109.175,-92.218,165.922,49.650,158.927
C02412=1021.744,-108.926,-92.227,165.925,49.646,158.927
C02413=1021.749,-108.676,-92.236,165.928,49.642,158.926
C02414=1021.755,-108.426,-92.245,165.932,49.638,158.926
C02415=1021.760,-108.176,-92.253,165.935,49.634,158.926
C02416=1021.766,-107.926,-92.261,165.938,49.631,158.926
C02417=1021.771,-107.677,-92.270,165.941,49.626,158.926
C02418=1021.777,-107.427,-92.280,165.943,49.622,158.925
C02419=1021.782,-107.177,-92.288,165.946,49.619,158.925
C02420=1021.788,-106.927,-92.296,165.950,49.615,158.925
C02421=1021.794,-106.677,-92.305,165.953,49.611,158.925
C02422=1021.799,-106.428,-92.315,165.956,49.607,158.925
C02423=1021.804,-106.178,-92.323,165.959,49.603,158.925
C02424=1021.810,-105.928,-92.332,165.962,49.600,158.925
C02425=1021.816,-105.678,-92.340,165.965,49.596,158.924
C02426=1021.821,-105.429,-92.350,165.969,49.592,158.924
C02427=1021.826,-105.179,-92.358,165.972,49.588,158.924
C02428=1021.831,-104.928,-92.367,165.974,49.584,158.924
C02429=1021.837,-104.679,-92.377,165.978,49.581,158.924
C02430=1021.842,-104.430,-92.385,165.980,49.577,158.923
C02431=1021.848,-104.179,-92.394,165.983,49.573,158.923
C02432=1021.854,-103.930,-92.403,165.987,49.569,158.923
C02433=1021.859,-103.680,-92.412,165.990,49.565,158.923
C02434=1021.865,-103.431,-92.421,165.993,49.562,158.923
C02435=1021.870,-103.181,-92.430,165.996,49.558,158.923
C02436=1021.876,-102.930,-92.439,165.999,49.554,158.922
C02437=1021.881,-102.681,-92.448,166.002,49.550,158.922
C02438=1021.886,-102.431,-92.457,166.004,49.546,158.922
C02439=1021.893,-102.182,-92.466,166.008,49.542,158.922
C02440=1021.898,-101.932,-92.475,166.011,49.539,158.922
C02441=1021.904,-101.646,-92.485,166.015,49.534,158.922
C02442=1021.911,-101.362,-92.496,166.018,49.530,158.921
C02443=1021.917,-101.077,-92.505,166.021,49.525,158.921
C02444=1021.923,-100.792,-92.516,166.025,49.521,158.921
C02445=1021.928,-100.542,-92.525,166.028,49.518,158.921
C02446=1021.935,-100.292,-92.535,166.031,49.514,158.920
C02447=1021.940,-100.042,-92.543,166.034,49.510,158.920
C02448=1021.945,-99.792,-92.553,166.038,49.506,158.920
C02449=1021.951,-99.542,-92.562,166.041,49.502,158.920
C02450=1021.957,-99.293,-92.571,166.044,49.498,158.920
C02451=1021.962,-99.044,-92.580,166.047,49.495,158.920
C02452=1021.968,-98.794,-92.589,166.049,49.491,158.919
C02453=1021.974,-98.544,-92.598,166.052,49.487,158.919
C02454=1021.978,-98.294,-92.608,166.056,49.483,158.919
C02455=1021.984,-98.044,-92.617,166.059,49.479,158.919
C02456=1021.990,-97.795,-92.626,166.062,49.475,158.919
C02457=1021.996,-97.545,-92.635,166.065,49.472,158.918
C02458=1022.001,-97.295,-92.645,166.068,49.468,158.918
C02459=1022.007,-97.045,-92.654,166.071,49.464,158.918
C02460=1022.012,-96.795,-92.664,166.074,49.460,158.918
C02461=1022.018,-96.546,-92.673,166.077,49.457,158.918
C02462=1022.023,-96.295,-92.682,166.081,49.453,158.918
C02463=1022.028,-96.046,-92.692,166.084,49.449,158.918
C02464=1022.034,-95.796,-92.701,166.086,49.445,158.917
C02465=1022.039,-95.547,-92.711,166.090,49.442,158.917
C02466=1022.045,-95.296,-92.720,166.092,49.438,158.917
C02467=1022.050,-95.047,-92.730,166.095,49.435,158.917
C02468=1022.056,-94.797,-92.739,166.098,49.431,158.917
C02469=1022.062,-94.548,-92.749,166.101,49.427,158.916
C02470=1022.067,-94.297,-92.758,166.104,49.423,158.916
C02471=1022.072,-94.048,-92.767,166.108,49.420,158.916
C02472=1022.078,-93.798,-92.777,166.111,49.416,158.916
C02473=1022.084,-93.548,-92.787,166.114,49.412,158.916
C02474=1022.089,-93.299,-92.797,166.117,49.408,158.916
C02475=1022.095,-93.048,-92.806,166.120,49.405,158.915
C02476=1022.100,-92.799,-92.815,166.123,49.401,158.915
C02477=1022.106,-92.549,-92.825,166.126,49.397,158.915
C02478=1022.111,-92.300,-92.834,166.129,49.394,158.915
C02479=1022.117,-92.050,-92.844,166.132,49.390,158.915
C02480=1022.123,-91.800,-92.854,166.136,49.386,158.915
C02481=1022.128,-91.551,-92.864,166.138,49.382,158.914
C02482=1022.134,-91.301,-92.873,166.142,49.379,158.914
C02483=1022.139,-91.050,-92.883,166.144,49.375,158.914
C02484=1022.145,-90.801,-92.892,166.147,49.371,158.914
C02485=1022.150,-90.551,-92.902,166.150,49.367,158.914
C02486=1022.156,-90.302,-92.911,166.153,49.363,158.913
C02487=1022.161,-90.052,-92.921,166.156,49.360,158.913
C02488=1022.167,-89.802,-92.931,166.160,49.356,158.913
C02489=1022.173,-89.553,-92.940,166.163,49.352,158.913
C02490=1022.178,-89.303,-92.950,166.166,49.348,158.913
C02491=1022.184,-89.053,-92.960,166.169,49.344,158.912
C02492=1022.189,-88.804,-92.970,166.172,49.341,158.912
C02493=1022.195,-88.554,-92.979,166.174,49.337,158.912
C02494=1022.201,-88.304,-92.989,166.178,49.334,158.912
C02495=1022.207,-88.054,-92.999,166.181,49.329,158.912
C02496=1022.212,-87.805,-93.009,166.184,49.325,158.912
C02497=1022.218,-87.555,-93.018,166.187,49.322,158.911
C02498=1022.223,-87.305,-93.029,166.190,49.318,158.911
C02499=1022.229,-87.056,-93.038,166.193,49.315,158.911
C02500=1022.234,-86.805,-93.048,166.196,49.311,158.911
C02501=1022.241,-86.556,-93.058,166.199,49.307,158.910
C02502=1022.246,-86.306,-93.068,166.203,49.303,158.911
C02503=1022.252,-86.056,-93.077,166.206,49.299,158.910
C02504=1022.257,-85.806,-93.087,166.208,49.295,158.910
C02505=1022.263,-85.523,-93.098,166.212,49.291,158.910
C02506=1022.271,-85.240,-93.109,166.215,49.287,158.910
C02507=1022.277,-84.958,-93.120,166.219,49.282,158.909
C02508=1022.283,-84.675,-93.131,166.223,49.278,158.909
C02509=1022.289,-84.425,-93.141,166.225,49.274,158.909
C02510=1022.295,-84.175,-93.151,166.229,49.271,158.909
C02511=1022.300,-83.925,-93.161,166.231,49.267,158.909
C02512=1022.306,-83.676,-93.170,166.234,49.263,158.908
C02513=1022.312,-83.427,-93.181,166.237,49.260,158.908
C02514=1022.318,-83.177,-93.191,166.241,49.255,158.908
C02515=1022.323,-82.927,-93.201,166.244,49.251,158.908
C02516=1022.329,-82.677,-93.211,166.247,49.247,158.907
C02517=1022.335,-82.427,-93.221,166.250,49.244,158.907
C02518=1022.340,-82.178,-93.230,166.253,49.240,158.907
C02519=1022.346,-81.928,-93.241,166.255,49.236,158.907
C02520=1022.352,-81.678,-93.250,166.260,49.232,158.907
C02521=1022.358,-81.428,-93.260,166.262,49.228,158.907
C02522=1022.364,-81.179,-93.270,166.265,49.224,158.906
C02523=1022.369,-80.928,-93.280,166.268,49.221,158.906
C02524=1022.376,-80.679,-93.290,166.271,49.217,158.906
C02525=1022.381,-80.430,-93.300,166.274,49.213,158.906
C02526=1022.387,-80.180,-93.310,166.278,49.209,158.905
C02527=1022.392,-79.930,-93.320,166.281,49.205,158.905
C02528=1022.398,-79.680,-93.331,166.283,49.201,158.905
C02529=1022.404,-79.430,-93.341,166.287,49.198,158.905
C02530=1022.410,-79.181,-93.351,166.289,49.194,158.905
C02531=1022.415,-78.931,-93.361,166.293,49.191,158.905
C02532=1022.421,-78.681,-93.372,166.295,49.187,158.904
C02533=1022.427,-78.431,-93.383,166.298,49.184,158.904
C02534=1022.433,-78.182,-93.392,166.301,49.180,158.904
C02535=1022.438,-77.933,-93.403,166.304,49.176,158.904
C02536=1022.443,-77.683,-93.413,166.307,49.172,158.904
C02537=1022.449,-77.433,-93.423,166.310,49.169,158.903
C02538=1022.455,-77.183,-93.434,166.314,49.165,158.903
C02539=1022.461,-76.933,-93.443,166.317,49.161,158.903
C02540=1022.466,-76.684,-93.454,166.320,49.157,158.903
C02541=1022.472,-76.434,-93.464,166.323,49.154,158.903
C02542=1022.478,-76.184,-93.475,166.326,49.150,158.902
C02543=1022.484,-75.934,-93.485,166.329,49.146,158.902
C02544=1022.490,-75.685,-93.496,166.332,49.143,158.902
C02545=1022.495,-75.435,-93.506,166.335,49.139,158.902
C02546=1022.501,-75.185,-93.517,166.337,49.135,158.902
C02547=1022.506,-74.935,-93.527,166.341,49.132,158.901
C02548=1022.513,-74.686,-93.537,166.344,49.127,158.901
C02549=1022.518,-74.436,-93.547,166.347,49.124,158.901
C02550=1022.524,-74.186,-93.558,166.350,49.120,158.901
C02551=1022.529,-73.936,-93.568,166.353,49.117,158.901
C02552=1022.535,-73.687,-93.579,166.356,49.113,158.900
C02553=1022.541,-73.437,-93.590,166.359,49.110,158.900
C02554=1022.546,-73.187,-93.600,166.362,49.106,158.900
C02555=1022.551,-72.937,-93.612,166.365,49.102,158.900
C02556=1022.557,-72.688,-93.623,166.368,49.099,158.900
C02557=1022.562,-72.438,-93.633,166.371,49.095,158.900
C02558=1022.568,-72.188,-93.644,166.374,49.092,158.899
C02559=1022.574,-71.939,-93.655,166.377,49.088,158.899
C02560=1022.580,-71.689,-93.665,166.380,49.084,158.899
C02561=1022.585,-71.439,-93.676,166.383,49.081,158.899
C02562=1022.591,-71.190,-93.687,166.386,49.077,158.899
C02563=1022.596,-70.940,-93.697,166.389,49.074,158.899
C02564=1022.602,-70.691,-93.708,166.392,49.070,158.898
C02565=1022.608,-70.441,-93.718,166.395,49.067,158.898
C02566=1022.613,-70.191,-93.729,166.398,49.063,158.898
C02567=1022.618,-69.941,-93.741,166.401,49.059,158.898
C02568=1022.624,-69.692,-93.752,166.404,49.056,158.898
C02569=1022.631,-69.410,-93.764,166.407,49.052,158.897
C02570=1022.638,-69.130,-93.776,166.411,49.048,158.897
C02571=1022.644,-68.849,-93.788,166.414,49.044,158.897
C02572=1022.650,-68.569,-93.800,166.417,49.040,158.897
C02573=1022.655,-68.318,-93.811,166.421,49.036,158.897
C02574=1022.661,-68.069,-93.822,166.423,49.032,158.896
C02575=1022.667,-67.819,-93.833,166.426,49.029,158.896
C02576=1022.673,-67.569,-93.844,166.429,49.025,158.896
C02577=1022.679,-67.320,-93.855,166.432,49.022,158.896
C02578=1022.684,-67.070,-93.866,166.435,49.018,158.896
C02579=1022.690,-66.821,-93.877,166.438,49.015,158.895
C02580=1022.696,-66.571,-93.887,166.441,49.011,158.895
C02581=1022.701,-66.321,-93.898,166.444,49.007,158.895
C02582=1022.707,-66.072,-93.908,166.447,49.003,158.895
C02583=1022.713,-65.821,-93.920,166.450,49.000,158.895
C02584=1022.718,-65.572,-93.931,166.453,48.996,158.894
C02585=1022.724,-65.322,-93.942,166.456,48.993,158.894
C02586=1022.730,-65.073,-93.953,166.459,48.989,158.894
C02587=1022.736,-64.823,-93.964,166.462,48.986,158.894
C02588=1022.741,-64.574,-93.975,166.465,48.982,158.894
C02589=1022.748,-64.323,-93.986,166.468,48.978,158.894
C02590=1022.753,-64.074,-93.997,166.471,48.974,158.893
C02591=1022.758,-63.824,-94.008,166.474,48.971,158.893
C02592=1022.764,-63.575,-94.019,166.477,48.967,158.893
C02593=1022.770,-63.325,-94.030,166.479,48.963,158.893
C02594=1022.776,-63.075,-94.041,166.483,48.960,158.892
C02595=1022.782,-62.825,-94.052,166.486,48.956,158.892
C02596=1022.788,-62.576,-94.063,166.490,48.952,158.892
C02597=1022.793,-62.327,-94.074,166.492,48.948,158.892
C02598=1022.800,-62.076,-94.085,166.495,48.945,158.892
C02599=1022.805,-61.827,-94.097,166.498,48.941,158.891
///RCONF 1,0,0,0,0,0,0,0,0,0,0,0,0,0,0,0,0,0,0,0,0,0,0,0
C02600=1022.811,-61.577,-94.107,166.501,48.938,158.891
C02601=1022.816,-61.328,-94.118,166.504,48.934,158.891
C02602=1022.823,-61.077,-94.130,166.507,48.930,158.891
C02603=1022.828,-60.828,-94.140,166.510,48.927,158.891
C02604=1022.834,-60.578,-94.151,166.513,48.923,158.890
C02605=1022.841,-60.329,-94.163,166.516,48.920,158.890
C02606=1022.847,-60.079,-94.174,166.519,48.916,158.890
C02607=1022.852,-59.830,-94.186,166.522,48.912,158.890
C02608=1022.858,-59.579,-94.197,166.525,48.908,158.890
C02609=1022.864,-59.330,-94.208,166.528,48.904,158.889
C02610=1022.869,-59.080,-94.219,166.531,48.901,158.889
C02611=1022.875,-58.831,-94.230,166.534,48.897,158.889
C02612=1022.881,-58.581,-94.241,166.536,48.893,158.889
C02613=1022.887,-58.331,-94.253,166.539,48.890,158.888
C02614=1022.892,-58.082,-94.264,166.542,48.886,158.888
C02615=1022.899,-57.832,-94.275,166.545,48.883,158.888
C02616=1022.905,-57.582,-94.286,166.548,48.879,158.888
C02617=1022.911,-57.332,-94.297,166.551,48.875,158.887
C02618=1022.917,-57.083,-94.308,166.555,48.871,158.887
C02619=1022.923,-56.834,-94.320,166.558,48.867,158.887
C02620=1022.928,-56.583,-94.332,166.561,48.863,158.887
C02621=1022.934,-56.334,-94.342,166.564,48.860,158.887
C02622=1022.940,-56.084,-94.353,166.567,48.856,158.886
C02623=1022.946,-55.835,-94.365,166.570,48.852,158.886
C02624=1022.952,-55.585,-94.376,166.573,48.849,158.886
C02625=1022.958,-55.335,-94.387,166.575,48.845,158.886
C02626=1022.963,-55.085,-94.399,166.578,48.841,158.885
C02627=1022.970,-54.836,-94.410,166.581,48.838,158.885
C02628=1022.976,-54.586,-94.422,166.584,48.834,158.885
C02629=1022.982,-54.337,-94.433,166.587,48.830,158.885
C02630=1022.988,-54.086,-94.444,166.590,48.827,158.885
C02631=1022.994,-53.838,-94.455,166.593,48.823,158.884
C02632=1023.000,-53.587,-94.467,166.596,48.819,158.884
C02633=1023.006,-53.308,-94.480,166.600,48.814,158.884
C02634=1023.013,-53.028,-94.492,166.602,48.810,158.884
C02635=1023.020,-52.748,-94.505,166.606,48.806,158.883
C02636=1023.027,-52.469,-94.518,166.610,48.802,158.883
C02637=1023.033,-52.219,-94.529,166.613,48.798,158.883
C02638=1023.039,-51.969,-94.541,166.616,48.794,158.883
C02639=1023.044,-51.720,-94.552,166.618,48.790,158.882
C02640=1023.051,-51.470,-94.564,166.622,48.787,158.882
C02641=1023.057,-51.221,-94.575,166.624,48.783,158.882
C02642=1023.063,-50.971,-94.586,166.627,48.779,158.882
C02643=1023.068,-50.721,-94.598,166.630,48.776,158.881
C02644=1023.075,-50.471,-94.610,166.633,48.772,158.881
C02645=1023.080,-50.222,-94.622,166.636,48.769,158.881
C02646=1023.086,-49.972,-94.634,166.639,48.765,158.881
C02647=1023.092,-49.723,-94.645,166.642,48.761,158.881
C02648=1023.097,-49.472,-94.657,166.645,48.757,158.880
C02649=1023.103,-49.223,-94.669,166.648,48.754,158.880
C02650=1023.109,-48.973,-94.681,166.650,48.750,158.880
C02651=1023.115,-48.724,-94.692,166.653,48.747,158.880
C02652=1023.121,-48.474,-94.705,166.656,48.744,158.880
C02653=1023.127,-48.225,-94.716,166.659,48.740,158.879
C02654=1023.133,-47.975,-94.728,166.662,48.737,158.879
C02655=1023.138,-47.726,-94.740,166.665,48.733,158.879
C02656=1023.144,-47.475,-94.752,166.668,48.730,158.879
C02657=1023.150,-47.226,-94.764,166.671,48.726,158.878
C02658=1023.156,-46.976,-94.775,166.674,48.722,158.878
C02659=1023.161,-46.727,-94.787,166.677,48.718,158.878
C02660=1023.168,-46.477,-94.799,166.680,48.715,158.878
C02661=1023.173,-46.227,-94.811,166.683,48.711,158.878
C02662=1023.179,-45.978,-94.823,166.686,48.707,158.877
C02663=1023.185,-45.728,-94.835,166.689,48.704,158.877
C02664=1023.191,-45.479,-94.847,166.692,48.700,158.877
C02665=1023.197,-45.229,-94.859,166.695,48.697,158.877
C02666=1023.202,-44.979,-94.871,166.698,48.693,158.876
C02667=1023.208,-44.730,-94.883,166.701,48.690,158.876
C02668=1023.215,-44.479,-94.895,166.704,48.686,158.876
C02669=1023.220,-44.230,-94.907,166.706,48.683,158.876
C02670=1023.227,-43.981,-94.919,166.708,48.679,158.876
C02671=1023.232,-43.731,-94.931,166.712,48.676,158.875
C02672=1023.237,-43.481,-94.943,166.714,48.672,158.875
C02673=1023.244,-43.231,-94.955,166.717,48.668,158.875
C02674=1023.249,-42.982,-94.967,166.720,48.665,158.875
C02675=1023.256,-42.733,-94.979,166.723,48.661,158.874
C02676=1023.262,-42.483,-94.991,166.726,48.657,158.874
C02677=1023.268,-42.233,-95.002,166.729,48.653,158.874
C02678=1023.274,-41.983,-95.015,166.732,48.650,158.874
C02679=1023.280,-41.733,-95.027,166.735,48.646,158.874
C02680=1023.286,-41.485,-95.039,166.738,48.642,158.873
C02681=1023.291,-41.235,-95.052,166.741,48.639,158.873
C02682=1023.297,-40.985,-95.064,166.744,48.635,158.873
C02683=1023.303,-40.735,-95.075,166.747,48.632,158.873
C02684=1023.309,-40.485,-95.088,166.750,48.628,158.872
C02685=1023.316,-40.236,-95.100,166.753,48.624,158.872
C02686=1023.321,-39.987,-95.112,166.756,48.621,158.872
C02687=1023.327,-39.737,-95.124,166.759,48.617,158.872
C02688=1023.334,-39.487,-95.136,166.761,48.613,158.871
C02689=1023.339,-39.237,-95.149,166.765,48.610,158.871
C02690=1023.345,-38.988,-95.161,166.766,48.606,158.871
C02691=1023.351,-38.739,-95.173,166.770,48.603,158.871
C02692=1023.357,-38.489,-95.186,166.772,48.599,158.870
C02693=1023.363,-38.239,-95.198,166.775,48.596,158.870
C02694=1023.369,-37.990,-95.210,166.778,48.592,158.870
C02695=1023.374,-37.740,-95.223,166.781,48.589,158.870
C02696=1023.380,-37.490,-95.235,166.785,48.585,158.870
C02697=1023.387,-37.211,-95.248,166.787,48.581,158.869
C02698=1023.393,-36.932,-95.263,166.790,48.577,158.869
C02699=1023.400,-36.652,-95.277,166.794,48.573,158.869
C02700=1023.407,-36.373,-95.291,166.797,48.569,158.869
C02701=1023.413,-36.123,-95.303,166.800,48.565,158.868
C02702=1023.418,-35.874,-95.315,166.803,48.562,158.868
C02703=1023.424,-35.624,-95.328,166.806,48.558,158.868
C02704=1023.430,-35.374,-95.341,166.809,48.555,158.868
C02705=1023.436,-35.124,-95.353,166.812,48.551,158.867
C02706=1023.442,-34.875,-95.365,166.814,48.548,158.867
C02707=1023.448,-34.626,-95.377,166.817,48.544,158.867
C02708=1023.454,-34.376,-95.391,166.820,48.541,158.867
C02709=1023.460,-34.126,-95.403,166.823,48.537,158.866
C02710=1023.466,-33.877,-95.416,166.826,48.534,158.866
C02711=1023.472,-33.627,-95.428,166.829,48.530,158.866
C02712=1023.477,-33.378,-95.440,166.832,48.527,158.866
C02713=1023.483,-33.128,-95.453,166.834,48.523,158.866
C02714=1023.489,-32.878,-95.466,166.838,48.520,158.865
C02715=1023.496,-32.629,-95.478,166.839,48.516,158.865
C02716=1023.502,-32.379,-95.491,166.843,48.513,158.865
C02717=1023.507,-32.129,-95.503,166.845,48.509,158.865
C02718=1023.513,-31.880,-95.515,166.848,48.505,158.864
C02719=1023.519,-31.631,-95.529,166.851,48.502,158.864
C02720=1023.525,-31.381,-95.541,166.854,48.498,158.864
C02721=1023.531,-31.131,-95.554,166.857,48.495,158.864
C02722=1023.537,-30.881,-95.566,166.860,48.491,158.863
C02723=1023.543,-30.632,-95.580,166.863,48.487,158.863
C02724=1023.550,-30.382,-95.592,166.865,48.484,158.863
C02725=1023.555,-30.133,-95.604,166.868,48.480,158.863
C02726=1023.561,-29.883,-95.616,166.871,48.477,158.862
C02727=1023.567,-29.634,-95.630,166.874,48.473,158.862
C02728=1023.573,-29.384,-95.642,166.877,48.470,158.862
C02729=1023.579,-29.134,-95.655,166.880,48.466,158.862
C02730=1023.585,-28.885,-95.668,166.883,48.462,158.861
C02731=1023.591,-28.635,-95.681,166.886,48.458,158.861
C02732=1023.597,-28.385,-95.693,166.889,48.455,158.861
C02733=1023.603,-28.136,-95.706,166.891,48.451,158.861
C02734=1023.609,-27.886,-95.719,166.894,48.448,158.860
C02735=1023.616,-27.636,-95.731,166.896,48.444,158.860
C02736=1023.622,-27.387,-95.744,166.900,48.441,158.860
C02737=1023.627,-27.137,-95.757,166.902,48.437,158.860
C02738=1023.632,-26.888,-95.770,166.906,48.433,158.860
C02739=1023.639,-26.638,-95.783,166.908,48.430,158.859
C02740=1023.644,-26.388,-95.795,166.911,48.427,158.859
C02741=1023.651,-26.139,-95.809,166.913,48.423,158.859
C02742=1023.657,-25.889,-95.821,166.916,48.420,158.859
C02743=1023.662,-25.640,-95.835,166.919,48.416,158.858
C02744=1023.668,-25.390,-95.848,166.922,48.412,158.858
C02745=1023.674,-25.141,-95.861,166.925,48.409,158.858
C02746=1023.680,-24.891,-95.873,166.927,48.406,158.858
C02747=1023.686,-24.641,-95.887,166.930,48.402,158.857
C02748=1023.692,-24.392,-95.901,166.933,48.398,158.857
C02749=1023.698,-24.142,-95.913,166.936,48.395,158.857
C02750=1023.704,-23.893,-95.926,166.939,48.391,158.857
C02751=1023.710,-23.643,-95.939,166.941,48.388,158.856
C02752=1023.716,-23.394,-95.952,166.944,48.385,158.856
C02753=1023.721,-23.143,-95.965,166.947,48.381,158.856
C02754=1023.727,-22.894,-95.979,166.950,48.377,158.856
C02755=1023.734,-22.645,-95.992,166.953,48.373,158.855
C02756=1023.740,-22.395,-96.004,166.956,48.370,158.855
C02757=1023.746,-22.146,-96.018,166.958,48.367,158.855
C02758=1023.752,-21.896,-96.030,166.961,48.363,158.855
C02759=1023.757,-21.646,-96.044,166.964,48.360,158.854
C02760=1023.763,-21.397,-96.057,166.967,48.356,158.854
C02761=1023.770,-21.116,-96.071,166.970,48.352,158.854
C02762=1023.777,-20.836,-96.086,166.973,48.349,158.854
C02763=1023.783,-20.556,-96.102,166.977,48.344,158.853
C02764=1023.791,-20.276,-96.116,166.980,48.340,158.853
C02765=1023.797,-20.026,-96.130,166.982,48.337,158.853
C02766=1023.803,-19.777,-96.142,166.985,48.333,158.853
C02767=1023.808,-19.527,-96.156,166.988,48.329,158.852
C02768=1023.814,-19.278,-96.169,166.990,48.326,158.852
C02769=1023.820,-19.028,-96.182,166.993,48.323,158.852
C02770=1023.826,-18.779,-96.195,166.996,48.319,158.852
C02771=1023.833,-18.529,-96.208,166.999,48.316,158.851
C02772=1023.838,-18.279,-96.222,167.002,48.312,158.851
C02773=1023.844,-18.030,-96.235,167.005,48.308,158.851
C02774=1023.851,-17.780,-96.248,167.007,48.305,158.851
C02775=1023.857,-17.531,-96.262,167.010,48.301,158.850
C02776=1023.863,-17.281,-96.274,167.013,48.297,158.850
C02777=1023.869,-17.031,-96.288,167.016,48.294,158.850
C02778=1023.875,-16.782,-96.301,167.019,48.290,158.849
C02779=1023.881,-16.533,-96.315,167.022,48.287,158.849
C02780=1023.887,-16.283,-96.327,167.024,48.283,158.849
C02781=1023.892,-16.033,-96.341,167.027,48.279,158.849
C02782=1023.899,-15.783,-96.355,167.030,48.276,158.848
C02783=1023.905,-15.534,-96.368,167.033,48.272,158.848
C02784=1023.911,-15.284,-96.382,167.036,48.269,158.848
C02785=1023.917,-15.035,-96.395,167.038,48.265,158.848
C02786=1023.923,-14.786,-96.409,167.041,48.262,158.847
C02787=1023.929,-14.536,-96.422,167.044,48.258,158.847
C02788=1023.935,-14.285,-96.436,167.047,48.255,158.847
C02789=1023.941,-14.036,-96.449,167.049,48.251,158.847
C02790=1023.946,-13.787,-96.463,167.052,48.248,158.846
C02791=1023.952,-13.537,-96.476,167.054,48.244,158.846
C02792=1023.958,-13.288,-96.490,167.058,48.241,158.846
C02793=1023.964,-13.038,-96.503,167.059,48.238,158.846
C02794=1023.970,-12.788,-96.518,167.063,48.234,158.845
C02795=1023.976,-12.539,-96.531,167.065,48.231,158.845
C02796=1023.982,-12.289,-96.545,167.069,48.227,158.845
C02797=1023.988,-12.040,-96.558,167.070,48.224,158.845
C02798=1023.994,-11.791,-96.572,167.074,48.221,158.844
C02799=1024.000,-11.541,-96.585,167.076,48.217,158.844
C02800=1024.007,-11.291,-96.599,167.080,48.213,158.844
C02801=1024.012,-11.042,-96.613,167.081,48.210,158.844
C02802=1024.018,-10.792,-96.626,167.085,48.207,158.843
C02803=1024.024,-10.542,-96.640,167.087,48.203,158.843
C02804=1024.031,-10.293,-96.653,167.090,48.199,158.843
C02805=1024.036,-10.043,-96.667,167.092,48.196,158.843
C02806=1024.043,-9.795,-96.681,167.095,48.192,158.842
C02807=1024.049,-9.544,-96.695,167.098,48.189,158.842
C02808=1024.055,-9.295,-96.709,167.101,48.185,158.842
C02809=1024.060,-9.046,-96.723,167.104,48.182,158.842
C02810=1024.067,-8.796,-96.736,167.106,48.178,158.841
C02811=1024.073,-8.546,-96.750,167.109,48.174,158.841
C02812=1024.079,-8.297,-96.763,167.112,48.171,158.841
C02813=1024.084,-8.047,-96.777,167.115,48.167,158.840
C02814=1024.091,-7.798,-96.791,167.117,48.164,158.840
C02815=1024.097,-7.548,-96.805,167.120,48.161,158.840
C02816=1024.102,-7.299,-96.819,167.123,48.157,158.840
C02817=1024.109,-7.049,-96.833,167.126,48.153,158.839
C02818=1024.115,-6.799,-96.847,167.128,48.150,158.839
C02819=1024.121,-6.550,-96.860,167.131,48.147,158.839
C02820=1024.126,-6.300,-96.874,167.134,48.143,158.839
C02821=1024.133,-6.050,-96.888,167.137,48.139,158.838
C02822=1024.139,-5.801,-96.902,167.140,48.136,158.838
C02823=1024.145,-5.552,-96.915,167.142,48.132,158.838
C02824=1024.151,-5.302,-96.930,167.144,48.128,158.837
C02825=1024.158,-5.020,-96.945,167.147,48.124,158.837
C02826=1024.165,-4.738,-96.961,167.151,48.120,158.837
C02827=1024.172,-4.457,-96.976,167.154,48.116,158.837
C02828=1024.179,-4.175,-96.992,167.157,48.112,158.836
C02829=1024.185,-3.925,-97.006,167.160,48.109,158.836
C02830=1024.190,-3.676,-97.020,167.163,48.105,158.836
C02831=1024.197,-3.426,-97.035,167.165,48.103,158.836
C02832=1024.202,-3.176,-97.048,167.168,48.099,158.835
C02833=1024.208,-2.927,-97.062,167.171,48.095,158.835
C02834=1024.214,-2.677,-97.077,167.173,48.092,158.835
C02835=1024.220,-2.428,-97.091,167.176,48.089,158.834
C02836=1024.226,-2.179,-97.105,167.179,48.085,158.834
C02837=1024.232,-1.929,-97.119,167.181,48.082,158.834
C02838=1024.238,-1.679,-97.133,167.184,48.078,158.834
C02839=1024.244,-1.429,-97.148,167.187,48.075,158.833
C02840=1024.250,-1.180,-97.162,167.189,48.072,158.833
C02841=1024.255,-0.931,-97.177,167.192,48.068,158.833
C02842=1024.262,-0.681,-97.190,167.195,48.065,158.833
C02843=1024.268,-0.432,-97.205,167.197,48.061,158.832
C02844=1024.273,-0.182,-97.219,167.200,48.058,158.832
C02845=1024.280,0.067,-97.234,167.203,48.054,158.832
C02846=1024.285,0.317,-97.247,167.205,48.051,158.832
C02847=1024.292,0.567,-97.262,167.208,48.048,158.831
C02848=1024.297,0.816,-97.276,167.211,48.044,158.831
C02849=1024.304,1.066,-97.291,167.213,48.041,158.831
C02850=1024.310,1.315,-97.305,167.216,48.038,158.831
C02851=1024.316,1.564,-97.319,167.219,48.034,158.830
C02852=1024.322,1.814,-97.333,167.221,48.031,158.830
C02853=1024.327,2.063,-97.348,167.224,48.027,158.830
C02854=1024.334,2.313,-97.362,167.227,48.024,158.830
C02855=1024.339,2.562,-97.377,167.229,48.020,158.829
C02856=1024.345,2.813,-97.391,167.232,48.016,158.829
C02857=1024.351,3.062,-97.406,167.235,48.013,158.829
C02858=1024.357,3.312,-97.420,167.237,48.010,158.828
C02859=1024.364,3.561,-97.434,167.240,48.006,158.828
C02860=1024.370,3.810,-97.448,167.243,48.003,158.828
C02861=1024.376,4.060,-97.463,167.245,48.000,158.828
C02862=1024.381,4.309,-97.477,167.248,47.996,158.827
C02863=1024.387,4.559,-97.491,167.251,47.993,158.827
C02864=1024.393,4.808,-97.506,167.254,47.989,158.827
C02865=1024.400,5.058,-97.521,167.256,47.985,158.826
C02866=1024.405,5.307,-97.535,167.259,47.982,158.826
C02867=1024.411,5.557,-97.550,167.262,47.978,158.826
C02868=1024.417,5.806,-97.564,167.264,47.975,158.826
C02869=1024.424,6.056,-97.578,167.267,47.971,158.825
C02870=1024.430,6.305,-97.593,167.270,47.968,158.825
C02871=1024.436,6.555,-97.607,167.272,47.965,158.825
C02872=1024.442,6.805,-97.622,167.275,47.961,158.824
C02873=1024.448,7.054,-97.636,167.278,47.958,158.824
C02874=1024.454,7.304,-97.650,167.280,47.954,158.824
C02875=1024.460,7.553,-97.665,167.282,47.950,158.824
C02876=1024.466,7.803,-97.680,167.286,47.947,158.823
C02877=1024.472,8.051,-97.695,167.288,47.943,158.823
C02878=1024.478,8.302,-97.709,167.291,47.940,158.823
C02879=1024.484,8.551,-97.723,167.293,47.937,158.822
C02880=1024.491,8.800,-97.738,167.296,47.933,158.822
C02881=1024.497,9.050,-97.752,167.298,47.930,158.822
C02882=1024.503,9.299,-97.767,167.301,47.926,158.822
C02883=1024.509,9.549,-97.782,167.304,47.922,158.821
C02884=1024.515,9.798,-97.796,167.306,47.919,158.821
C02885=1024.521,10.048,-97.810,167.309,47.915,158.821
C02886=1024.527,10.297,-97.825,167.312,47.911,158.820
C02887=1024.533,10.547,-97.840,167.315,47.908,158.820
C02888=1024.540,10.796,-97.855,167.317,47.905,158.820
C02889=1024.547,11.080,-97.871,167.320,47.901,158.819
C02890=1024.554,11.363,-97.888,167.324,47.897,158.819
C02891=1024.560,11.647,-97.904,167.326,47.892,158.819
C02892=1024.568,11.931,-97.921,167.329,47.888,158.818
C02893=1024.574,12.180,-97.936,167.332,47.885,158.818
C02894=1024.580,12.431,-97.950,167.334,47.882,158.818
C02895=1024.586,12.680,-97.965,167.337,47.878,158.818
C02896=1024.592,12.929,-97.980,167.340,47.874,158.817
C02897=1024.598,13.179,-97.994,167.343,47.871,158.817
C02898=1024.604,13.428,-98.009,167.345,47.867,158.817
C02899=1024.611,13.678,-98.024,167.348,47.863,158.816
C02900=1024.617,13.927,-98.039,167.351,47.860,158.816
C02901=1024.623,14.176,-98.053,167.353,47.857,158.816
C02902=1024.629,14.426,-98.068,167.356,47.854,158.816
C02903=1024.635,14.676,-98.083,167.358,47.850,158.815
C02904=1024.640,14.925,-98.098,167.361,47.847,158.815
C02905=1024.647,15.175,-98.113,167.364,47.843,158.815
C02906=1024.653,15.425,-98.128,167.366,47.839,158.814
C02907=1024.659,15.674,-98.142,167.369,47.836,158.814
C02908=1024.665,15.923,-98.158,167.372,47.832,158.814
C02909=1024.671,16.173,-98.174,167.374,47.830,158.814
C02910=1024.677,16.422,-98.188,167.377,47.826,158.813
C02911=1024.683,16.671,-98.203,167.379,47.822,158.813
C02912=1024.690,16.921,-98.218,167.382,47.819,158.813
C02913=1024.695,17.170,-98.233,167.385,47.815,158.812
C02914=1024.701,17.420,-98.248,167.387,47.812,158.812
C02915=1024.707,17.669,-98.263,167.390,47.808,158.812
C02916=1024.714,17.919,-98.278,167.392,47.805,158.811
C02917=1024.720,18.168,-98.293,167.395,47.802,158.811
C02918=1024.726,18.418,-98.308,167.397,47.798,158.811
C02919=1024.732,18.668,-98.323,167.401,47.795,158.811
C02920=1024.737,18.917,-98.338,167.402,47.791,158.810
C02921=1024.744,19.166,-98.353,167.405,47.787,158.810
C02922=1024.750,19.416,-98.368,167.408,47.784,158.810
C02923=1024.756,19.665,-98.384,167.410,47.781,158.809
C02924=1024.762,19.914,-98.398,167.413,47.777,158.809
C02925=1024.768,20.164,-98.413,167.415,47.774,158.809
C02926=1024.774,20.414,-98.429,167.418,47.770,158.808
C02927=1024.780,20.664,-98.444,167.421,47.767,158.808
C02928=1024.786,20.912,-98.460,167.423,47.763,158.808
C02929=1024.792,21.162,-98.475,167.426,47.760,158.808
C02930=1024.798,21.412,-98.490,167.428,47.757,158.807
C02931=1024.804,21.661,-98.505,167.431,47.754,158.807
C02932=1024.810,21.910,-98.520,167.434,47.750,158.807
C02933=1024.817,22.159,-98.535,167.436,47.746,158.806
C02934=1024.822,22.409,-98.551,167.439,47.743,158.806
C02935=1024.829,22.659,-98.566,167.441,47.739,158.806
C02936=1024.834,22.908,-98.580,167.444,47.736,158.806
C02937=1024.840,23.157,-98.597,167.447,47.732,158.805
C02938=1024.847,23.407,-98.612,167.449,47.729,158.805
C02939=1024.852,23.657,-98.627,167.452,47.726,158.805
C02940=1024.859,23.906,-98.643,167.455,47.722,158.804
C02941=1024.865,24.155,-98.657,167.457,47.719,158.804
C02942=1024.870,24.405,-98.673,167.460,47.715,158.804
C02943=1024.877,24.655,-98.688,167.462,47.712,158.803
C02944=1024.884,24.904,-98.704,167.465,47.709,158.803
C02945=1024.889,25.154,-98.719,167.468,47.705,158.803
C02946=1024.896,25.403,-98.734,167.470,47.701,158.802
C02947=1024.901,25.652,-98.750,167.473,47.698,158.802
C02948=1024.907,25.902,-98.765,167.475,47.694,158.802
C02949=1024.914,26.151,-98.780,167.478,47.691,158.802
C02950=1024.920,26.401,-98.796,167.481,47.688,158.801
C02951=1024.926,26.650,-98.811,167.483,47.684,158.801
C02952=1024.932,26.900,-98.827,167.486,47.681,158.801
C02953=1024.939,27.185,-98.844,167.488,47.676,158.800
C02954=1024.946,27.470,-98.862,167.491,47.673,158.800
C02955=1024.952,27.755,-98.879,167.494,47.669,158.800
C02956=1024.960,28.040,-98.897,167.497,47.665,158.799
C02957=1024.966,28.289,-98.913,167.500,47.661,158.799
C02958=1024.971,28.539,-98.929,167.502,47.658,158.799
C02959=1024.978,28.788,-98.945,167.505,47.654,158.798
C02960=1024.983,29.038,-98.960,167.508,47.651,158.798
C02961=1024.990,29.287,-98.975,167.510,47.648,158.798
C02962=1024.996,29.537,-98.991,167.513,47.645,158.798
C02963=1025.001,29.786,-99.007,167.515,47.641,158.797
C02964=1025.008,30.036,-99.022,167.518,47.637,158.797
C02965=1025.014,30.285,-99.038,167.520,47.634,158.797
C02966=1025.020,30.535,-99.053,167.523,47.631,158.796
C02967=1025.026,30.784,-99.070,167.526,47.627,158.796
C02968=1025.031,31.033,-99.085,167.528,47.624,158.796
C02969=1025.038,31.282,-99.101,167.531,47.621,158.796
C02970=1025.044,31.532,-99.116,167.533,47.617,158.795
C02971=1025.049,31.782,-99.132,167.536,47.613,158.795
C02972=1025.056,32.031,-99.148,167.538,47.610,158.795
C02973=1025.062,32.281,-99.164,167.541,47.607,158.794
C02974=1025.068,32.530,-99.179,167.544,47.603,158.794
C02975=1025.074,32.780,-99.195,167.546,47.600,158.794
C02976=1025.080,33.029,-99.211,167.549,47.596,158.793
C02977=1025.087,33.278,-99.227,167.551,47.593,158.793
C02978=1025.092,33.528,-99.242,167.554,47.590,158.793
C02979=1025.098,33.777,-99.258,167.557,47.586,158.792
C02980=1025.105,34.026,-99.274,167.559,47.583,158.792
C02981=1025.111,34.276,-99.290,167.562,47.579,158.792
C02982=1025.117,34.525,-99.305,167.564,47.575,158.791
C02983=1025.123,34.775,-99.322,167.567,47.572,158.791
C02984=1025.128,35.024,-99.337,167.569,47.569,158.791
C02985=1025.135,35.273,-99.352,167.572,47.565,158.790
C02986=1025.141,35.522,-99.369,167.575,47.562,158.790
C02987=1025.147,35.772,-99.384,167.577,47.558,158.790
C02988=1025.153,36.021,-99.400,167.579,47.555,158.789
C02989=1025.163,36.435,-99.427,167.584,47.549,158.789
C02990=1025.174,36.848,-99.452,167.588,47.543,158.788
C02991=1025.184,37.261,-99.479,167.592,47.537,158.788
C02992=1025.194,37.675,-99.505,167.596,47.532,158.787
C02993=1025.200,37.925,-99.521,167.599,47.529,158.787
C02994=1025.206,38.174,-99.538,167.601,47.525,158.787
C02995=1025.212,38.423,-99.554,167.604,47.522,158.787
C02996=1025.218,38.673,-99.570,167.607,47.518,158.786
C02997=1025.224,38.922,-99.586,167.609,47.516,158.786
C02998=1025.229,39.171,-99.603,167.612,47.512,158.786
C02999=1025.235,39.421,-99.618,167.614,47.508,158.785
C03000=1025.242,39.670,-99.634,167.617,47.505,158.785
C03001=1025.248,39.920,-99.650,167.619,47.502,158.785
C03002=1025.254,40.169,-99.666,167.622,47.498,158.785
C03003=1025.260,40.418,-99.683,167.624,47.495,158.784
C03004=1025.266,40.668,-99.699,167.627,47.492,158.784
C03005=1025.272,40.917,-99.715,167.629,47.488,158.783
C03006=1025.278,41.166,-99.731,167.632,47.484,158.783
C03007=1025.283,41.416,-99.748,167.635,47.481,158.783
C03008=1025.290,41.665,-99.763,167.637,47.478,158.783
C03009=1025.296,41.915,-99.779,167.640,47.474,158.782
C03010=1025.302,42.165,-99.796,167.642,47.471,158.782
C03011=1025.308,42.414,-99.812,167.645,47.467,158.782
C03012=1025.314,42.664,-99.828,167.647,47.465,158.781
C03013=1025.323,43.034,-99.853,167.650,47.459,158.781
C03014=1025.332,43.405,-99.877,167.655,47.454,158.780
C03015=1025.341,43.775,-99.901,167.658,47.449,158.780
C03016=1025.350,44.146,-99.926,167.662,47.445,158.780
C03017=1025.356,44.395,-99.942,167.664,47.441,158.779
C03018=1025.361,44.645,-99.959,167.667,47.438,158.779
C03019=1025.367,44.894,-99.975,167.669,47.434,158.779
C03020=1025.373,45.143,-99.992,167.672,47.431,158.778
C03021=1025.379,45.393,-100.008,167.674,47.428,158.778
C03022=1025.385,45.642,-100.024,167.677,47.425,158.778
C03023=1025.391,45.891,-100.040,167.679,47.421,158.777
C03024=1025.396,46.140,-100.058,167.682,47.418,158.777
C03025=1025.402,46.390,-100.074,167.684,47.415,158.777
C03026=1025.409,46.640,-100.091,167.687,47.411,158.777
C03027=1025.415,46.889,-100.107,167.689,47.408,158.776
C03028=1025.421,47.139,-100.123,167.692,47.405,158.776
C03029=1025.426,47.388,-100.140,167.694,47.401,158.776
C03030=1025.432,47.637,-100.157,167.697,47.398,158.775
C03031=1025.438,47.886,-100.173,167.699,47.395,158.775
C03032=1025.444,48.136,-100.190,167.702,47.392,158.775
C03033=1025.450,48.386,-100.206,167.704,47.388,158.774
C03034=1025.456,48.635,-100.223,167.708,47.385,158.774
C03035=1025.463,48.884,-100.240,167.709,47.381,158.774
C03036=1025.468,49.133,-100.256,167.712,47.378,158.773
C03037=1025.474,49.383,-100.273,167.714,47.375,158.773
C03038=1025.480,49.632,-100.289,167.717,47.371,158.773
C03039=1025.486,49.881,-100.306,167.720,47.368,158.773
C03040=1025.493,50.131,-100.322,167.722,47.364,158.772
C03041=1025.499,50.380,-100.339,167.725,47.362,158.772
C03042=1025.504,50.630,-100.356,167.727,47.358,158.772
C03043=1025.510,50.879,-100.373,167.729,47.354,158.771
C03044=1025.516,51.128,-100.389,167.733,47.351,158.771
C03045=1025.523,51.378,-100.405,167.734,47.348,158.771
C03046=1025.528,51.627,-100.422,167.738,47.345,158.770
C03047=1025.534,51.876,-100.439,167.739,47.341,158.770
C03048=1025.540,52.126,-100.456,167.742,47.337,158.770
C03049=1025.546,52.375,-100.472,167.745,47.334,158.769
C03050=1025.553,52.624,-100.489,167.747,47.331,158.769
C03051=1025.559,52.874,-100.505,167.751,47.328,158.769
C03052=1025.564,53.124,-100.522,167.752,47.324,158.768
C03053=1025.570,53.372,-100.539,167.755,47.320,158.768
C03054=1025.577,53.622,-100.556,167.758,47.317,158.768
C03055=1025.583,53.872,-100.572,167.760,47.314,158.768
C03056=1025.589,54.120,-100.589,167.762,47.310,158.767
C03057=1025.594,54.370,-100.606,167.766,47.307,158.767
C03058=1025.601,54.620,-100.623,167.767,47.303,158.766
C03059=1025.607,54.869,-100.639,167.770,47.300,158.766
C03060=1025.613,55.118,-100.656,167.772,47.297,158.766
C03061=1025.619,55.367,-100.673,167.775,47.293,158.766
C03062=1025.625,55.617,-100.690,167.777,47.290,158.765
C03063=1025.631,55.867,-100.706,167.780,47.286,158.765
C03064=1025.637,56.115,-100.723,167.782,47.283,158.765
C03065=1025.643,56.365,-100.739,167.785,47.279,158.764
C03066=1025.650,56.614,-100.757,167.788,47.276,158.764
C03067=1025.655,56.864,-100.774,167.790,47.273,158.764
C03068=1025.661,57.113,-100.790,167.793,47.269,158.763
C03069=1025.668,57.363,-100.807,167.795,47.266,158.763
C03070=1025.674,57.612,-100.823,167.798,47.262,158.763
C03071=1025.680,57.861,-100.840,167.800,47.259,158.762
C03072=1025.686,58.111,-100.858,167.803,47.255,158.762
C03073=1025.692,58.360,-100.875,167.805,47.252,158.762
C03074=1025.698,58.609,-100.891,167.808,47.248,158.761
C03075=1025.705,58.858,-100.908,167.811,47.245,158.761
C03076=1025.711,59.108,-100.924,167.813,47.242,158.761
C03077=1025.717,59.393,-100.944,167.816,47.237,158.760
C03078=1025.725,59.677,-100.964,167.819,47.234,158.760
C03079=1025.732,59.962,-100.983,167.822,47.230,158.759
C03080=1025.739,60.247,-101.002,167.824,47.225,158.759
C03081=1025.745,60.496,-101.019,167.827,47.222,158.759
C03082=1025.751,60.746,-101.036,167.830,47.218,158.758
C03083=1025.757,60.995,-101.053,167.832,47.215,158.758
C03084=1025.763,61.244,-101.069,167.835,47.211,158.758
C03085=1025.770,61.494,-101.087,167.837,47.208,158.757
C03086=1025.775,61.743,-101.103,167.840,47.205,158.757
C03087=1025.782,61.993,-101.121,167.842,47.201,158.757
C03088=1025.788,62.242,-101.137,167.845,47.197,158.756
C03089=1025.794,62.491,-101.154,167.848,47.194,158.756
C03090=1025.801,62.741,-101.171,167.850,47.191,158.756
C03091=1025.807,62.990,-101.188,167.853,47.187,158.755
C03092=1025.813,63.239,-101.205,167.855,47.183,158.755
C03093=1025.819,63.489,-101.222,167.858,47.180,158.755
C03094=1025.825,63.738,-101.239,167.860,47.177,158.754
C03095=1025.831,63.988,-101.257,167.863,47.173,158.754
C03096=1025.837,64.237,-101.273,167.865,47.170,158.754
C03097=1025.843,64.487,-101.291,167.868,47.167,158.753
C03098=1025.849,64.735,-101.308,167.870,47.164,158.753
C03099=1025.855,64.985,-101.325,167.873,47.160,158.753
C03100=1025.861,65.234,-101.343,167.875,47.156,158.752
C03101=1025.867,65.483,-101.360,167.878,47.153,158.752
C03102=1025.874,65.733,-101.377,167.880,47.150,158.752
C03103=1025.879,65.982,-101.395,167.883,47.146,158.751
C03104=1025.886,66.232,-101.412,167.885,47.143,158.751
C03105=1025.891,66.481,-101.429,167.888,47.140,158.751
C03106=1025.898,66.730,-101.446,167.890,47.136,158.750
C03107=1025.904,66.980,-101.464,167.893,47.133,158.750
C03108=1025.909,67.229,-101.482,167.895,47.130,158.750
C03109=1025.916,67.479,-101.498,167.898,47.126,158.749
C03110=1025.921,67.728,-101.516,167.900,47.123,158.749
C03111=1025.928,67.977,-101.533,167.903,47.119,158.749
C03112=1025.934,68.226,-101.551,167.906,47.116,158.748
C03113=1025.940,68.475,-101.568,167.908,47.113,158.748
C03114=1025.946,68.725,-101.586,167.911,47.109,158.748
C03115=1025.951,68.974,-101.603,167.913,47.106,158.747
C03116=1025.958,69.224,-101.620,167.916,47.102,158.747
C03117=1025.964,69.473,-101.637,167.918,47.099,158.747
C03118=1025.970,69.722,-101.655,167.921,47.096,158.746
C03119=1025.975,69.972,-101.673,167.923,47.092,158.746
C03120=1025.982,70.221,-101.690,167.926,47.089,158.746
C03121=1025.988,70.470,-101.708,167.928,47.086,158.745
C03122=1025.994,70.720,-101.726,167.930,47.083,158.745
C03123=1026.000,70.968,-101.743,167.933,47.079,158.745
C03124=1026.006,71.218,-101.761,167.935,47.076,158.744
C03125=1026.012,71.467,-101.778,167.938,47.073,158.744
C03126=1026.018,71.717,-101.796,167.940,47.069,158.744
C03127=1026.024,71.966,-101.813,167.943,47.066,158.744
C03128=1026.030,72.215,-101.831,167.945,47.063,158.743
C03129=1026.036,72.464,-101.849,167.948,47.059,158.743
C03130=1026.042,72.714,-101.867,167.950,47.056,158.743
C03131=1026.048,72.963,-101.884,167.953,47.052,158.742
C03132=1026.054,73.213,-101.902,167.955,47.049,158.742
C03133=1026.060,73.462,-101.919,167.958,47.046,158.742
C03134=1026.066,73.711,-101.937,167.960,47.042,158.741
C03135=1026.071,73.961,-101.955,167.963,47.039,158.741
C03136=1026.078,74.210,-101.972,167.966,47.035,158.741
C03137=1026.084,74.459,-101.989,167.968,47.032,158.740
C03138=1026.090,74.709,-102.007,167.971,47.029,158.740
C03139=1026.095,74.958,-102.025,167.973,47.025,158.740
C03140=1026.102,75.207,-102.042,167.976,47.022,158.739
C03141=1026.109,75.492,-102.063,167.979,47.018,158.739
C03142=1026.116,75.776,-102.083,167.982,47.014,158.738
C03143=1026.122,76.061,-102.103,167.985,47.010,158.738
C03144=1026.130,76.345,-102.123,167.988,47.007,158.738
C03145=1026.136,76.594,-102.142,167.990,47.003,158.737
C03146=1026.142,76.844,-102.160,167.993,46.999,158.737
C03147=1026.148,77.093,-102.177,167.995,46.997,158.737
C03148=1026.154,77.343,-102.195,167.998,46.993,158.736
C03149=1026.159,77.592,-102.213,168.000,46.990,158.736
C03150=1026.165,77.842,-102.231,168.003,46.986,158.736
C03151=1026.171,78.090,-102.249,168.005,46.984,158.735
C03152=1026.177,78.340,-102.267,168.008,46.980,158.735
C03153=1026.184,78.590,-102.285,168.010,46.976,158.735
C03154=1026.189,78.839,-102.302,168.013,46.973,158.735
C03155=1026.195,79.088,-102.321,168.015,46.970,158.734
C03156=1026.201,79.337,-102.338,168.017,46.967,158.734
C03157=1026.207,79.587,-102.356,168.020,46.963,158.733
C03158=1026.213,79.835,-102.375,168.022,46.960,158.733
C03159=1026.219,80.085,-102.393,168.025,46.957,158.733
C03160=1026.225,80.334,-102.411,168.027,46.954,158.733
C03161=1026.231,80.583,-102.429,168.030,46.950,158.732
C03162=1026.237,80.833,-102.447,168.032,46.947,158.732
C03163=1026.243,81.082,-102.464,168.035,46.944,158.732
C03164=1026.249,81.331,-102.483,168.037,46.940,158.731
C03165=1026.254,81.581,-102.501,168.040,46.937,158.731
C03166=1026.260,81.830,-102.519,168.042,46.934,158.731
C03167=1026.266,82.079,-102.538,168.046,46.931,158.730
C03168=1026.273,82.329,-102.556,168.047,46.927,158.730
C03169=1026.278,82.578,-102.573,168.051,46.924,158.730
C03170=1026.284,82.827,-102.592,168.053,46.921,158.729
C03171=1026.290,83.076,-102.609,168.055,46.917,158.729
C03172=1026.296,83.325,-102.628,168.058,46.914,158.729
C03173=1026.303,83.575,-102.646,168.061,46.910,158.728
C03174=1026.308,83.824,-102.664,168.063,46.908,158.728
C03175=1026.314,84.073,-102.682,168.066,46.904,158.728
C03176=1026.321,84.323,-102.700,168.068,46.900,158.727
C03177=1026.326,84.571,-102.718,168.071,46.897,158.727
C03178=1026.333,84.821,-102.736,168.073,46.894,158.727
C03179=1026.339,85.071,-102.754,168.076,46.890,158.726
C03180=1026.344,85.319,-102.773,168.078,46.887,158.726
C03181=1026.351,85.569,-102.790,168.081,46.884,158.726
C03182=1026.356,85.818,-102.810,168.083,46.881,158.725
C03183=1026.362,86.068,-102.828,168.086,46.877,158.725
C03184=1026.368,86.316,-102.846,168.088,46.874,158.725
C03185=1026.374,86.566,-102.864,168.091,46.871,158.724
C03186=1026.381,86.815,-102.883,168.094,46.867,158.724
C03187=1026.386,87.064,-102.900,168.096,46.863,158.724
C03188=1026.393,87.313,-102.919,168.099,46.860,158.723
C03189=1026.399,87.563,-102.937,168.101,46.857,158.723
C03190=1026.405,87.812,-102.955,168.104,46.853,158.723
C03191=1026.411,88.061,-102.973,168.106,46.850,158.722
C03192=1026.417,88.310,-102.992,168.109,46.847,158.722
C03193=1026.423,88.560,-103.009,168.111,46.843,158.722
C03194=1026.430,88.809,-103.028,168.114,46.840,158.721
C03195=1026.435,89.058,-103.046,168.116,46.837,158.721
C03196=1026.441,89.308,-103.065,168.119,46.833,158.721
C03197=1026.447,89.557,-103.084,168.121,46.830,158.720
C03198=1026.454,89.807,-103.102,168.124,46.826,158.720
C03199=1026.459,90.055,-103.120,168.126,46.824,158.720
C03200=1026.465,90.305,-103.138,168.129,46.820,158.719
C03201=1026.471,90.554,-103.157,168.131,46.817,158.719
C03202=1026.477,90.804,-103.176,168.134,46.813,158.719
C03203=1026.482,91.053,-103.194,168.136,46.811,158.718
C03204=1026.489,91.302,-103.212,168.139,46.807,158.718
C03205=1026.495,91.586,-103.234,168.142,46.803,158.718
C03206=1026.503,91.871,-103.255,168.145,46.799,158.717
C03207=1026.509,92.156,-103.276,168.148,46.796,158.717
C03208=1026.516,92.440,-103.298,168.151,46.792,158.717
C03209=1026.521,92.689,-103.317,168.153,46.789,158.716
C03210=1026.528,92.938,-103.335,168.156,46.786,158.716
C03211=1026.534,93.188,-103.353,168.158,46.782,158.716
C03212=1026.539,93.437,-103.372,168.161,46.779,158.715
C03213=1026.545,93.686,-103.391,168.163,46.776,158.715
C03214=1026.552,93.935,-103.409,168.166,46.773,158.715
C03215=1026.557,94.185,-103.428,168.168,46.769,158.714
C03216=1026.563,94.434,-103.447,168.171,46.765,158.714
C03217=1026.569,94.683,-103.466,168.174,46.763,158.714
C03218=1026.575,94.932,-103.484,168.176,46.759,158.713
C03219=1026.581,95.181,-103.503,168.179,46.756,158.713
C03220=1026.587,95.431,-103.521,168.182,46.752,158.713
C03221=1026.593,95.680,-103.540,168.184,46.750,158.712
C03222=1026.599,95.930,-103.559,168.187,46.746,158.712
C03223=1026.605,96.179,-103.578,168.190,46.742,158.712
C03224=1026.611,96.427,-103.596,168.192,46.739,158.711
C03225=1026.617,96.677,-103.615,168.195,46.736,158.711
C03226=1026.623,96.926,-103.633,168.197,46.733,158.711
C03227=1026.629,97.175,-103.652,168.200,46.729,158.710
C03228=1026.635,97.425,-103.671,168.202,46.726,158.710
C03229=1026.642,97.674,-103.690,168.205,46.723,158.710
C03230=1026.647,97.923,-103.709,168.207,46.719,158.709
C03231=1026.653,98.172,-103.727,168.210,46.716,158.709
C03232=1026.659,98.421,-103.746,168.212,46.713,158.709
C03233=1026.665,98.670,-103.765,168.215,46.709,158.708
C03234=1026.672,98.920,-103.784,168.218,46.706,158.708
C03235=1026.677,99.170,-103.802,168.220,46.703,158.708
C03236=1026.683,99.419,-103.821,168.223,46.699,158.707
C03237=1026.690,99.668,-103.840,168.225,46.696,158.707
C03238=1026.695,99.917,-103.859,168.228,46.692,158.707
C03239=1026.701,100.167,-103.878,168.230,46.690,158.706
C03240=1026.707,100.415,-103.896,168.233,46.686,158.706
C03241=1026.713,100.665,-103.916,168.236,46.683,158.706
C03242=1026.718,100.914,-103.935,168.238,46.679,158.705
C03243=1026.725,101.163,-103.954,168.241,46.677,158.705
C03244=1026.731,101.412,-103.974,168.244,46.673,158.705
C03245=1026.736,101.661,-103.993,168.246,46.670,158.705
C03246=1026.743,101.910,-104.011,168.249,46.667,158.704
C03247=1026.749,102.160,-104.031,168.251,46.664,158.704
C03248=1026.754,102.409,-104.050,168.254,46.660,158.704
C03249=1026.759,102.658,-104.069,168.256,46.657,158.703
C03250=1026.766,102.907,-104.087,168.259,46.654,158.703
C03251=1026.771,103.157,-104.107,168.261,46.651,158.703
C03252=1026.777,103.406,-104.126,168.264,46.647,158.702
C03253=1026.784,103.655,-104.145,168.266,46.644,158.702
C03254=1026.790,103.904,-104.165,168.269,46.641,158.702
C03255=1026.795,104.153,-104.184,168.272,46.638,158.701
C03256=1026.802,104.403,-104.202,168.274,46.634,158.701
C03257=1026.807,104.652,-104.222,168.277,46.631,158.701
C03258=1026.813,104.901,-104.241,168.280,46.628,158.700
C03259=1026.820,105.150,-104.260,168.283,46.625,158.700
C03260=1026.826,105.399,-104.280,168.285,46.621,158.700
C03261=1026.831,105.649,-104.299,168.288,46.618,158.700
C03262=1026.838,105.898,-104.317,168.290,46.615,158.699
C03263=1026.843,106.147,-104.337,168.293,46.612,158.699
C03264=1026.849,106.397,-104.356,168.295,46.608,158.698
C03265=1026.856,106.645,-104.375,168.298,46.605,158.698
C03266=1026.861,106.895,-104.394,168.300,46.602,158.698
C03267=1026.867,107.144,-104.414,168.303,46.598,158.697
C03268=1026.873,107.394,-104.433,168.305,46.595,158.697
C03269=1026.880,107.677,-104.455,168.309,46.591,158.697
C03270=1026.887,107.962,-104.477,168.312,46.588,158.696
C03271=1026.894,108.247,-104.499,168.315,46.584,158.696
C03272=1026.901,108.532,-104.521,168.318,46.580,158.696
C03273=1026.907,108.781,-104.541,168.320,46.577,158.695
C03274=1026.912,109.030,-104.560,168.323,46.573,158.695
C03275=1026.919,109.279,-104.578,168.325,46.571,158.695
C03276=1026.925,109.528,-104.598,168.328,46.567,158.694
C03277=1026.930,109.778,-104.618,168.331,46.564,158.694
C03278=1026.937,110.027,-104.636,168.333,46.560,158.694
C03279=1026.943,110.275,-104.656,168.337,46.557,158.693
C03280=1026.949,110.525,-104.676,168.338,46.554,158.693
C03281=1026.954,110.774,-104.695,168.342,46.551,158.693
C03282=1026.960,111.023,-104.715,168.344,46.548,158.692
C03283=1026.966,111.273,-104.734,168.347,46.545,158.692
C03284=1026.972,111.522,-104.753,168.350,46.541,158.692
C03285=1026.978,111.771,-104.773,168.352,46.538,158.692
C03286=1026.984,112.020,-104.792,168.355,46.534,158.691
C03287=1026.990,112.269,-104.812,168.357,46.531,158.691
C03288=1026.996,112.518,-104.831,168.360,46.528,158.691
C03289=1027.002,112.767,-104.851,168.362,46.525,158.690
C03290=1027.007,113.016,-104.870,168.365,46.522,158.690
C03291=1027.013,113.265,-104.890,168.367,46.519,158.690
C03292=1027.018,113.515,-104.910,168.370,46.515,158.689
C03293=1027.025,113.764,-104.930,168.373,46.512,158.689
C03294=1027.031,114.014,-104.950,168.376,46.509,158.689
C03295=1027.037,114.263,-104.970,168.378,46.506,158.688
C03296=1027.043,114.512,-104.990,168.381,46.503,158.688
C03297=1027.048,114.761,-105.009,168.383,46.500,158.688
C03298=1027.054,115.010,-105.029,168.386,46.496,158.687
C03299=1027.059,115.260,-105.049,168.389,46.493,158.687
C03300=1027.065,115.508,-105.069,168.391,46.490,158.687
C03301=1027.071,115.757,-105.088,168.395,46.487,158.687
C03302=1027.077,116.007,-105.108,168.397,46.484,158.686
C03303=1027.083,116.255,-105.128,168.400,46.481,158.686
C03304=1027.089,116.504,-105.148,168.402,46.478,158.686
C03305=1027.094,116.754,-105.167,168.405,46.474,158.685
C03306=1027.100,117.003,-105.187,168.407,46.471,158.685
C03307=1027.106,117.252,-105.208,168.410,46.468,158.685
C03308=1027.112,117.502,-105.227,168.412,46.465,158.684
C03309=1027.118,117.751,-105.247,168.415,46.462,158.684
C03310=1027.124,117.999,-105.267,168.417,46.459,158.684
C03311=1027.129,118.249,-105.287,168.421,46.456,158.684
C03312=1027.135,118.498,-105.307,168.424,46.453,158.683
C03313=1027.141,118.747,-105.327,168.426,46.449,158.683
C03314=1027.147,118.996,-105.346,168.429,46.446,158.683
C03315=1027.153,119.246,-105.366,168.431,46.443,158.682
C03316=1027.159,119.494,-105.386,168.434,46.440,158.682
C03317=1027.165,119.744,-105.407,168.436,46.437,158.682
C03318=1027.170,119.993,-105.426,168.439,46.433,158.681
C03319=1027.176,120.242,-105.446,168.443,46.430,158.681
C03320=1027.182,120.491,-105.466,168.445,46.427,158.681
C03321=1027.188,120.739,-105.486,168.448,46.424,158.681
C03322=1027.194,120.990,-105.505,168.450,46.420,158.680
C03323=1027.200,121.239,-105.526,168.453,46.417,158.680
C03324=1027.206,121.488,-105.546,168.455,46.414,158.679
C03325=1027.212,121.736,-105.566,168.458,46.411,158.679
C03326=1027.218,121.985,-105.586,168.461,46.408,158.679
C03327=1027.224,122.235,-105.606,168.463,46.405,158.679
C03328=1027.229,122.484,-105.626,168.466,46.402,158.678
C03329=1027.235,122.733,-105.646,168.468,46.398,158.678
C03330=1027.241,122.982,-105.666,168.472,46.395,158.678
C03331=1027.247,123.231,-105.686,168.475,46.392,158.677
C03332=1027.254,123.480,-105.706,168.477,46.389,158.677
C03333=1027.260,123.765,-105.730,168.480,46.385,158.677
C03334=1027.267,124.050,-105.752,168.484,46.381,158.676
C03335=1027.274,124.335,-105.775,168.487,46.378,158.676
C03336=1027.281,124.619,-105.798,168.490,46.374,158.676
C03337=1027.287,124.868,-105.817,168.493,46.371,158.675
C03338=1027.293,125.117,-105.837,168.495,46.368,158.675
C03339=1027.298,125.366,-105.858,168.498,46.365,158.675
C03340=1027.305,125.615,-105.878,168.500,46.361,158.674
C03341=1027.310,125.864,-105.898,168.503,46.358,158.674
C03342=1027.316,126.113,-105.918,168.506,46.355,158.674
C03343=1027.322,126.362,-105.938,168.508,46.352,158.673
C03344=1027.328,126.612,-105.959,168.511,46.348,158.673
C03345=1027.334,126.860,-105.979,168.515,46.345,158.673
C03346=1027.340,127.109,-105.999,168.517,46.342,158.672
C03347=1027.347,127.359,-106.019,168.520,46.339,158.672
C03348=1027.353,127.608,-106.039,168.523,46.335,158.672
C03349=1027.358,127.857,-106.059,168.525,46.332,158.672
C03350=1027.364,128.106,-106.079,168.528,46.329,158.671
C03351=1027.370,128.356,-106.099,168.531,46.326,158.671
C03352=1027.376,128.604,-106.119,168.533,46.322,158.671
C03353=1027.382,128.854,-106.140,168.536,46.319,158.670
C03354=1027.388,129.103,-106.160,168.539,46.316,158.670
C03355=1027.394,129.352,-106.180,168.542,46.313,158.670
C03356=1027.401,129.600,-106.201,168.544,46.309,158.669
C03357=1027.407,129.850,-106.221,168.548,46.306,158.669
C03358=1027.412,130.099,-106.242,168.550,46.303,158.669
C03359=1027.419,130.348,-106.262,168.553,46.300,158.668
C03360=1027.425,130.597,-106.282,168.556,46.296,158.668
C03361=1027.430,130.846,-106.303,168.558,46.294,158.668
C03362=1027.437,131.096,-106.323,168.561,46.291,158.668
C03363=1027.442,131.345,-106.344,168.564,46.287,158.667
C03364=1027.448,131.593,-106.365,168.566,46.284,158.667
C03365=1027.454,131.842,-106.385,168.570,46.281,158.667
C03366=1027.460,132.092,-106.406,168.572,46.278,158.666
C03367=1027.466,132.341,-106.426,168.575,46.275,158.666
C03368=1027.471,132.591,-106.447,168.578,46.272,158.666
C03369=1027.478,132.839,-106.467,168.580,46.268,158.665
C03370=1027.483,133.088,-106.488,168.583,46.265,158.665
C03371=1027.490,133.337,-106.508,168.587,46.262,158.665
C03372=1027.495,133.587,-106.529,168.589,46.259,158.665
C03373=1027.501,133.835,-106.549,168.592,46.256,158.664
C03374=1027.507,134.085,-106.570,168.595,46.253,158.664
C03375=1027.513,134.333,-106.590,168.597,46.250,158.664
C03376=1027.518,134.583,-106.611,168.600,46.247,158.663
C03377=1027.524,134.832,-106.632,168.603,46.244,158.663
C03378=1027.530,135.081,-106.652,168.605,46.240,158.663
C03379=1027.536,135.330,-106.673,168.609,46.237,158.663
C03380=1027.543,135.579,-106.694,168.612,46.234,158.662
C03381=1027.548,135.828,-106.715,168.614,46.231,158.662
C03382=1027.554,136.077,-106.735,168.617,46.228,158.662
C03383=1027.560,136.326,-106.756,168.620,46.225,158.661
C03384=1027.566,136.576,-106.777,168.622,46.222,158.661
C03385=1027.572,136.824,-106.797,168.625,46.219,158.661
C03386=1027.578,137.074,-106.819,168.629,46.216,158.661
C03387=1027.583,137.323,-106.839,168.631,46.212,158.660
C03388=1027.590,137.571,-106.860,168.634,46.209,158.660
C03389=1027.595,137.821,-106.881,168.637,46.206,158.660
C03390=1027.601,138.070,-106.901,168.639,46.203,158.659
C03391=1027.608,138.319,-106.922,168.642,46.200,158.659
C03392=1027.613,138.568,-106.943,168.646,46.197,158.659
C03393=1027.620,138.817,-106.964,168.648,46.194,158.658
C03394=1027.625,139.066,-106.985,168.651,46.191,158.658
C03395=1027.631,139.315,-107.006,168.654,46.188,158.658
C03396=1027.636,139.564,-107.027,168.656,46.185,158.658
C03397=1027.643,139.848,-107.051,168.660,46.181,158.657
C03398=1027.650,140.132,-107.075,168.663,46.177,158.657
C03399=1027.657,140.417,-107.099,168.666,46.175,158.657
C03400=1027.664,140.702,-107.122,168.669,46.171,158.656
C03401=1027.669,140.950,-107.144,168.673,46.168,158.656
C03402=1027.675,141.199,-107.165,168.676,46.164,158.656
C03403=1027.680,141.449,-107.186,168.678,46.162,158.656
C03404=1027.687,141.698,-107.207,168.681,46.159,158.655
C03405=1027.693,141.947,-107.227,168.684,46.156,158.655
C03406=1027.699,142.196,-107.249,168.686,46.152,158.655
C03407=1027.704,142.444,-107.270,168.690,46.149,158.654
C03408=1027.710,142.694,-107.291,168.693,46.146,158.654
C03409=1027.716,142.943,-107.313,168.695,46.144,158.654
C03410=1027.722,143.192,-107.333,168.698,46.140,158.654
C03411=1027.728,143.441,-107.354,168.701,46.137,158.653
C03412=1027.734,143.690,-107.376,168.704,46.134,158.653
C03413=1027.739,143.939,-107.396,168.706,46.131,158.653
C03414=1027.746,144.188,-107.418,168.710,46.128,158.652
C03415=1027.751,144.437,-107.439,168.713,46.125,158.652
C03416=1027.758,144.686,-107.460,168.715,46.122,158.652
C03417=1027.763,144.935,-107.481,168.718,46.118,158.652
C03418=1027.769,145.184,-107.502,168.721,46.115,158.651
C03419=1027.775,145.434,-107.523,168.725,46.112,158.651
C03420=1027.781,145.682,-107.545,168.727,46.110,158.651
C03421=1027.787,145.931,-107.566,168.730,46.106,158.650
C03422=1027.793,146.180,-107.587,168.733,46.103,158.650
C03423=1027.799,146.429,-107.608,168.736,46.100,158.650
C03424=1027.805,146.678,-107.629,168.739,46.098,158.650
C03425=1027.811,146.927,-107.651,168.741,46.094,158.649
C03426=1027.817,147.176,-107.672,168.745,46.091,158.649
C03427=1027.823,147.425,-107.694,168.748,46.088,158.649
C03428=1027.828,147.675,-107.715,168.750,46.085,158.649
C03429=1027.834,147.923,-107.736,168.753,46.082,158.648
C03430=1027.840,148.172,-107.757,168.757,46.079,158.648
C03431=1027.846,148.422,-107.780,168.759,46.076,158.648
C03432=1027.851,148.670,-107.801,168.762,46.073,158.648
C03433=1027.857,148.920,-107.823,168.765,46.070,158.647
C03434=1027.863,149.168,-107.844,168.768,46.067,158.647
C03435=1027.869,149.417,-107.866,168.771,46.064,158.647
C03436=1027.875,149.667,-107.887,168.774,46.061,158.647
C03437=1027.880,149.916,-107.908,168.777,46.058,158.646
C03438=1027.887,150.165,-107.929,168.780,46.055,158.646
C03439=1027.892,150.413,-107.951,168.782,46.052,158.646
C03440=1027.898,150.663,-107.972,168.786,46.049,158.645
C03441=1027.905,150.912,-107.994,168.789,46.046,158.645
C03442=1027.910,151.160,-108.015,168.792,46.043,158.645
C03443=1027.916,151.410,-108.037,168.794,46.041,158.645
C03444=1027.922,151.659,-108.059,168.797,46.037,158.644
C03445=1027.927,151.908,-108.080,168.801,46.034,158.644
C03446=1027.933,152.157,-108.102,168.804,46.031,158.644
C03447=1027.940,152.406,-108.124,168.806,46.028,158.644
C03448=1027.945,152.654,-108.145,168.809,46.025,158.643
C03449=1027.951,152.904,-108.166,168.813,46.023,158.643
C03450=1027.957,153.153,-108.188,168.816,46.019,158.643
C03451=1027.963,153.401,-108.209,168.819,46.016,158.643
C03452=1027.969,153.650,-108.232,168.821,46.013,158.642
C03453=1027.975,153.899,-108.254,168.824,46.010,158.642
C03454=1027.980,154.148,-108.275,168.828,46.007,158.642
C03455=1027.987,154.397,-108.297,168.831,46.004,158.642
C03456=1027.993,154.646,-108.318,168.833,46.002,158.641
C03457=1027.998,154.896,-108.341,168.836,45.999,158.641
C03458=1028.004,155.144,-108.362,168.839,45.996,158.641
C03459=1028.010,155.394,-108.384,168.843,45.993,158.641
C03460=1028.016,155.642,-108.406,168.846,45.989,158.640
C03461=1028.022,155.927,-108.431,168.849,45.986,158.640
C03462=1028.029,156.210,-108.456,168.852,45.983,158.640
C03463=1028.036,156.495,-108.480,168.856,45.980,158.640
C03464=1028.042,156.779,-108.506,168.859,45.976,158.639
C03465=1028.048,157.028,-108.527,168.862,45.973,158.639
C03466=1028.055,157.277,-108.550,168.866,45.970,158.639
C03467=1028.060,157.525,-108.571,168.868,45.967,158.638
C03468=1028.066,157.775,-108.593,168.871,45.964,158.638
C03469=1028.072,158.024,-108.615,168.874,45.961,158.638
C03470=1028.079,158.272,-108.637,168.878,45.959,158.638
C03471=1028.083,158.521,-108.659,168.881,45.956,158.637
C03472=1028.090,158.770,-108.681,168.883,45.953,158.637
C03473=1028.096,159.020,-108.702,168.886,45.950,158.637
C03474=1028.102,159.268,-108.725,168.890,45.947,158.637
C03475=1028.108,159.518,-108.747,168.893,45.944,158.637
C03476=1028.113,159.766,-108.768,168.896,45.941,158.636
C03477=1028.119,160.015,-108.791,168.898,45.938,158.636
C03478=1028.124,160.265,-108.813,168.902,45.936,158.636
C03479=1028.130,160.514,-108.836,168.905,45.933,158.636
C03480=1028.136,160.762,-108.857,168.908,45.930,158.635
C03481=1028.141,161.011,-108.880,168.910,45.927,158.635
C03482=1028.147,161.260,-108.903,168.914,45.925,158.635
C03483=1028.153,161.509,-108.925,168.917,45.922,158.635
C03484=1028.158,161.758,-108.947,168.920,45.919,158.635
C03485=1028.164,162.007,-108.970,168.924,45.916,158.634
C03486=1028.170,162.255,-108.992,168.926,45.913,158.634
C03487=1028.176,162.505,-109.014,168.929,45.910,158.634
C03488=1028.181,162.753,-109.037,168.932,45.907,158.634
C03489=1028.186,163.003,-109.059,168.936,45.905,158.633
C03490=1028.193,163.251,-109.081,168.938,45.902,158.633
C03491=1028.198,163.501,-109.104,168.941,45.899,158.633
C03492=1028.204,163.750,-109.127,168.945,45.896,158.633
C03493=1028.210,163.998,-109.149,168.948,45.894,158.633
C03494=1028.215,164.247,-109.171,168.951,45.891,158.632
C03495=1028.221,164.496,-109.194,168.955,45.888,158.632
C03496=1028.227,164.745,-109.217,168.957,45.886,158.632
C03497=1028.233,164.994,-109.238,168.960,45.883,158.632
C03498=1028.238,165.243,-109.261,168.964,45.880,158.631
C03499=1028.244,165.492,-109.284,168.967,45.877,158.631
C03500=1028.250,165.740,-109.306,168.970,45.874,158.631
C03501=1028.256,165.989,-109.329,168.973,45.871,158.631
C03502=1028.261,166.238,-109.351,168.976,45.869,158.631
C03503=1028.267,166.488,-109.374,168.979,45.866,158.630
C03504=1028.273,166.736,-109.396,168.982,45.863,158.630
C03505=1028.279,166.985,-109.419,168.986,45.860,158.630
C03506=1028.284,167.235,-109.441,168.989,45.857,158.630
C03507=1028.290,167.483,-109.464,168.992,45.854,158.630
C03508=1028.296,167.732,-109.487,168.994,45.852,158.629
C03509=1028.302,167.980,-109.509,168.998,45.849,158.629
C03510=1028.307,168.230,-109.531,169.001,45.846,158.629
C03511=1028.314,168.478,-109.554,169.004,45.844,158.629
C03512=1028.319,168.727,-109.577,169.008,45.841,158.628
C03513=1028.325,168.976,-109.600,169.011,45.838,158.628
C03514=1028.330,169.226,-109.622,169.014,45.835,158.628
C03515=1028.337,169.474,-109.644,169.017,45.832,158.628
C03516=1028.343,169.723,-109.667,169.021,45.830,158.628
C03517=1028.348,169.972,-109.690,169.023,45.827,158.627
C03518=1028.354,170.221,-109.713,169.026,45.824,158.627
C03519=1028.361,170.470,-109.735,169.030,45.821,158.627
C03520=1028.366,170.719,-109.758,169.033,45.818,158.627
C03521=1028.372,170.968,-109.781,169.036,45.815,158.627
C03522=1028.377,171.217,-109.803,169.040,45.813,158.626
C03523=1028.384,171.465,-109.826,169.043,45.810,158.626
C03524=1028.390,171.714,-109.849,169.046,45.807,158.626
C03525=1028.396,171.998,-109.874,169.050,45.804,158.626
C03526=1028.403,172.282,-109.900,169.054,45.800,158.625
C03527=1028.410,172.565,-109.926,169.057,45.797,158.625
C03528=1028.417,172.849,-109.952,169.061,45.794,158.625
C03529=1028.422,173.098,-109.975,169.064,45.791,158.625
C03530=1028.428,173.347,-109.998,169.068,45.788,158.625
C03531=1028.434,173.596,-110.020,169.071,45.786,158.624
C03532=1028.440,173.845,-110.043,169.074,45.783,158.624
C03533=1028.446,174.094,-110.066,169.078,45.780,158.624
C03534=1028.452,174.343,-110.089,169.081,45.777,158.624
C03535=1028.458,174.591,-110.112,169.083,45.775,158.623
C03536=1028.464,174.840,-110.135,169.086,45.772,158.623
C03537=1028.470,175.089,-110.157,169.090,45.770,158.623
C03538=1028.475,175.338,-110.180,169.093,45.767,158.623
C03539=1028.481,175.587,-110.203,169.096,45.764,158.623
C03540=1028.488,175.835,-110.226,169.100,45.761,158.622
C03541=1028.493,176.084,-110.249,169.103,45.758,158.622
C03542=1028.500,176.334,-110.272,169.106,45.755,158.622
C03543=1028.505,176.583,-110.295,169.110,45.753,158.622
C03544=1028.512,176.831,-110.317,169.113,45.750,158.622
C03545=1028.518,177.080,-110.340,169.116,45.747,158.621
C03546=1028.524,177.328,-110.364,169.120,45.744,158.621
C03547=1028.529,177.577,-110.387,169.123,45.741,158.621
C03548=1028.535,177.826,-110.410,169.126,45.739,158.621
C03549=1028.542,178.076,-110.433,169.130,45.736,158.621
C03550=1028.548,178.324,-110.455,169.134,45.733,158.621
C03551=1028.554,178.573,-110.478,169.137,45.730,158.620
C03552=1028.559,178.822,-110.501,169.140,45.727,158.620
C03553=1028.566,179.071,-110.524,169.144,45.725,158.620
C03554=1028.572,179.320,-110.548,169.147,45.722,158.620
C03555=1028.578,179.569,-110.571,169.150,45.719,158.620
C03556=1028.584,179.818,-110.594,169.154,45.716,158.619
C03557=1028.590,180.066,-110.617,169.157,45.713,158.619
C03558=1028.596,180.315,-110.639,169.161,45.711,158.619
C03559=1028.603,180.564,-110.663,169.164,45.708,158.619
C03560=1028.608,180.813,-110.686,169.167,45.705,158.619
C03561=1028.614,181.062,-110.709,169.170,45.702,158.618
C03562=1028.620,181.311,-110.732,169.174,45.699,158.618
C03563=1028.627,181.560,-110.754,169.177,45.697,158.618
C03564=1028.633,181.808,-110.778,169.180,45.694,158.618
C03565=1028.639,182.057,-110.801,169.184,45.691,158.618
C03566=1028.644,182.306,-110.824,169.188,45.688,158.617
C03567=1028.651,182.555,-110.848,169.191,45.685,158.617
C03568=1028.658,182.804,-110.870,169.195,45.683,158.617
C03569=1028.663,183.053,-110.894,169.198,45.680,158.617
C03570=1028.669,183.301,-110.918,169.201,45.678,158.617
C03571=1028.674,183.550,-110.941,169.205,45.675,158.616
C03572=1028.680,183.799,-110.965,169.208,45.673,158.616
C03573=1028.686,184.048,-110.989,169.212,45.670,158.616
C03574=1028.691,184.297,-111.012,169.215,45.667,158.616
C03575=1028.697,184.545,-111.036,169.218,45.665,158.616
C03576=1028.702,184.794,-111.060,169.222,45.662,158.616
C03577=1028.709,185.043,-111.084,169.225,45.660,158.616
C03578=1028.715,185.292,-111.107,169.229,45.657,158.615
C03579=1028.720,185.541,-111.131,169.232,45.655,158.615
C03580=1028.726,185.789,-111.154,169.235,45.652,158.615
C03581=1028.732,186.039,-111.178,169.239,45.650,158.615
C03582=1028.738,186.287,-111.202,169.242,45.647,158.615
C03583=1028.744,186.535,-111.226,169.246,45.645,158.615
C03584=1028.749,186.785,-111.249,169.249,45.642,158.615
C03585=1028.755,187.034,-111.273,169.253,45.640,158.614
C03586=1028.761,187.282,-111.298,169.256,45.637,158.614
C03587=1028.766,187.531,-111.320,169.259,45.634,158.614
C03588=1028.773,187.780,-111.345,169.263,45.632,158.614
C03589=1028.779,188.063,-111.372,169.267,45.629,158.614
C03590=1028.786,188.347,-111.399,169.270,45.626,158.614
C03591=1028.792,188.630,-111.426,169.275,45.623,158.613
C03592=1028.799,188.913,-111.453,169.279,45.621,158.613
C03593=1028.805,189.162,-111.478,169.283,45.618,158.613
C03594=1028.810,189.411,-111.500,169.286,45.615,158.613
C03595=1028.817,189.660,-111.525,169.289,45.612,158.613
C03596=1028.822,189.908,-111.549,169.293,45.610,158.613
C03597=1028.828,190.156,-111.572,169.296,45.608,158.613
C03598=1028.834,190.406,-111.597,169.300,45.605,158.613
